LIN {X 0,Y 119.872,Z 1061.457,A -85,B 0,C 180,E1 -25663.563,E2 -25663.563} C_VEL
LIN {X 0,Y 121.874,Z 1058.966,A -85,B 0,C 180,E1 -25670.242,E2 -25670.242} C_VEL
LIN {X 0,Y 125.218,Z 1055.451,A -85,B 0,C 180,E1 -25676.679,E2 -25676.679} C_VEL
LIN {X 0,Y 129.866,Z 1050.86,A -85,B 0,C 180,E1 -25682.763,E2 -25682.763} C_VEL
LIN {X 0,Y 135.81,Z 1045.124,A -85,B 0,C 180,E1 -25688.387,E2 -25688.387} C_VEL
LIN {X 0,Y 141.031,Z 1040.06,A -85,B 0,C 180,E1 -25692.278,E2 -25692.278} C_VEL
LIN {X 0,Y 148.928,Z 1032.029,A -85,B 0,C 180,E1 -25697.007,E2 -25697.007} C_VEL
LIN {X 0,Y 151.068,Z 1029.838,A -85,B 0,C 180,E1 -25698.076,E2 -25698.076} C_VEL
LIN {X 0,Y 153.644,Z 1026.725,A -85,B 0,C 180,E1 -25699.683,E2 -25699.683} C_VEL
LIN {X 0,Y 156.483,Z 1021.432,A -85,B 0,C 180,E1 -25702.602,E2 -25702.602} C_VEL
LIN {X 0,Y 159.483,Z 1015.894,A -85,B 0,C 180,E1 -25705.377,E2 -25705.377} C_VEL
LIN {X 0,Y 162.214,Z 1012.21,A -85,B 0,C 180,E1 -25706.721,E2 -25706.721} C_VEL
LIN {X 0,Y 171.119,Z 1001.077,A -85,B 0,C 180,E1 -25709.594,E2 -25709.594} C_VEL
LIN {X 0,Y 180.348,Z 987.934,A -85,B 0,C 180,E1 -25712.119,E2 -25712.119} C_VEL
LIN {X 0,Y 187.112,Z 977.199,A -85,B 0,C 180,E1 -25713.732,E2 -25713.732} C_VEL
LIN {X 0,Y 193.609,Z 965.54,A -85,B 0,C 180,E1 -25715.158,E2 -25715.158} C_VEL
LIN {X 0,Y 199.505,Z 953.526,A -85,B 0,C 180,E1 -25716.331,E2 -25716.331} C_VEL
LIN {X 0,Y 204.688,Z 941.214,A -85,B 0,C 180,E1 -25717.329,E2 -25717.329} C_VEL
LIN {X 0,Y 209.238,Z 928.68,A -85,B 0,C 180,E1 -25718.103,E2 -25718.103} C_VEL
LIN {X 0,Y 213.187,Z 915.532,A -85,B 0,C 180,E1 -25718.738,E2 -25718.738} C_VEL
LIN {X 0,Y 216.353,Z 902.36,A -85,B 0,C 180,E1 -25719.211,E2 -25719.211} C_VEL
LIN {X 0,Y 218.607,Z 889.44,A -85,B 0,C 180,E1 -25719.615,E2 -25719.615} C_VEL
LIN {X 0,Y 221.458,Z 863.499,A -85,B 0,C 180,E1 -25720.238,E2 -25720.238} C_VEL
LIN {X 0,Y 225.126,Z 826.857,A -85,B 0,C 180,E1 -25721.038,E2 -25721.038} C_VEL
LIN {X 0,Y 223.867,Z 823.253,A -85,B 0,C 180,E1 -25722.353,E2 -25722.353} C_VEL
LIN {X 0,Y 221.348,Z 817.719,A -85,B 0,C 180,E1 -25725.167,E2 -25725.167} C_VEL
LIN {X 0,Y 219.032,Z 813.003,A -85,B 0,C 180,E1 -25728.334,E2 -25728.334} C_VEL
LIN {X 0,Y 217.674,Z 810.199,A -85,B 0,C 180,E1 -25730.709,E2 -25730.709} C_VEL
LIN {X 0,Y 216.21,Z 806.853,A -85,B 0,C 180,E1 -25734.403,E2 -25734.403} C_VEL
LIN {X 0,Y 215.341,Z 804.93,A -85,B 0,C 180,E1 -25739.999,E2 -25739.999} C_VEL
LIN {X 0,Y 216.416,Z 807.28,A -85,B 0,C 180,E1 -25746.643,E2 -25746.643} C_VEL
LIN {X 0,Y 218.274,Z 811.333,A -85,B 0,C 180,E1 -25750.797,E2 -25750.797} C_VEL
LIN {X 0,Y 220.254,Z 815.508,A -85,B 0,C 180,E1 -25753.845,E2 -25753.845} C_VEL
LIN {X 0,Y 222.437,Z 820.088,A -85,B 0,C 180,E1 -25756.52,E2 -25756.52} C_VEL
LIN {X 0,Y 226.001,Z 828.064,A -85,B 0,C 180,E1 -25760.109,E2 -25760.109} C_VEL
LIN {X 0,Y 234.508,Z 846.019,A -85,B 0,C 180,E1 -25766.47,E2 -25766.47} C_VEL
LIN {X 0,Y 241.894,Z 856.796,A -85,B 0,C 180,E1 -25770.446,E2 -25770.446} C_VEL
LIN {X 0,Y 249.216,Z 865.395,A -85,B 0,C 180,E1 -25773.663,E2 -25773.663} C_VEL
LIN {X 0,Y 263.908,Z 879.329,A -85,B 0,C 180,E1 -25778.879,E2 -25778.879} C_VEL
LIN {X 0,Y 280.399,Z 892.407,A -85,B 0,C 180,E1 -25783.707,E2 -25783.707} C_VEL
LIN {X 0,Y 288.067,Z 898.214,A -85,B 0,C 180,E1 -25786.03,E2 -25786.03} C_VEL
LIN {X 0,Y 295.771,Z 904.316,A -85,B 0,C 180,E1 -25788.563,E2 -25788.563} C_VEL
LIN {X 0,Y 302.153,Z 909.232,A -85,B 0,C 180,E1 -25790.793,E2 -25790.793} C_VEL
LIN {X 0,Y 308.739,Z 914.279,A -85,B 0,C 180,E1 -25793.23,E2 -25793.23} C_VEL
LIN {X 0,Y 315.739,Z 919.877,A -85,B 0,C 180,E1 -25796.013,E2 -25796.013} C_VEL
LIN {X 0,Y 322.198,Z 924.602,A -85,B 0,C 180,E1 -25798.709,E2 -25798.709} C_VEL
LIN {X 0,Y 327.662,Z 928.89,A -85,B 0,C 180,E1 -25801.207,E2 -25801.207} C_VEL
LIN {X 0,Y 332.858,Z 932.301,A -85,B 0,C 180,E1 -25803.68,E2 -25803.68} C_VEL
LIN {X 0,Y 337.92,Z 936.346,A -85,B 0,C 180,E1 -25806.391,E2 -25806.391} C_VEL
LIN {X 0,Y 341.187,Z 938.576,A -85,B 0,C 180,E1 -25808.237,E2 -25808.237} C_VEL
LIN {X 0,Y 345.175,Z 940.955,A -85,B 0,C 180,E1 -25810.656,E2 -25810.656} C_VEL
LIN {X 0,Y 348.889,Z 944.049,A -85,B 0,C 180,E1 -25813.398,E2 -25813.398} C_VEL
LIN {X 0,Y 352.119,Z 946.467,A -85,B 0,C 180,E1 -25816.143,E2 -25816.143} C_VEL
LIN {X 0,Y 354.613,Z 947.948,A -85,B 0,C 180,E1 -25818.569,E2 -25818.569} C_VEL
LIN {X 0,Y 356.684,Z 948.845,A -85,B 0,C 180,E1 -25820.931,E2 -25820.931} C_VEL
LIN {X 0,Y 358.262,Z 949.527,A -85,B 0,C 180,E1 -25823.241,E2 -25823.241} C_VEL
LIN {X 0,Y 359.416,Z 950.168,A -85,B 0,C 180,E1 -25825.741,E2 -25825.741} C_VEL
LIN {X 0,Y 360.008,Z 950.332,A -85,B 0,C 180,E1 -25827.762,E2 -25827.762} C_VEL
LIN {X 0,Y 360.177,Z 950.528,A -85,B 0,C 180,E1 -25830,E2 -25830} C_VEL
LIN {X 0,Y 359.997,Z 950.345,A -85,B 0,C 180,E1 -25832.238,E2 -25832.238} C_VEL
LIN {X 0,Y 359.347,Z 950.13,A -85,B 0,C 180,E1 -25834.487,E2 -25834.487} C_VEL
LIN {X 0,Y 358.254,Z 949.537,A -85,B 0,C 180,E1 -25836.759,E2 -25836.759} C_VEL
LIN {X 0,Y 356.317,Z 948.732,A -85,B 0,C 180,E1 -25839.534,E2 -25839.534} C_VEL
LIN {X 0,Y 353.687,Z 947.457,A -85,B 0,C 180,E1 -25842.357,E2 -25842.357} C_VEL
LIN {X 0,Y 350.683,Z 945.481,A -85,B 0,C 180,E1 -25845.101,E2 -25845.101} C_VEL
LIN {X 0,Y 347.397,Z 942.776,A -85,B 0,C 180,E1 -25847.758,E2 -25847.758} C_VEL
LIN {X 0,Y 345.062,Z 940.837,A -85,B 0,C 180,E1 -25849.424,E2 -25849.424} C_VEL
LIN {X 0,Y 340.899,Z 938.445,A -85,B 0,C 180,E1 -25851.919,E2 -25851.919} C_VEL
LIN {X 0,Y 335.973,Z 934.874,A -85,B 0,C 180,E1 -25854.67,E2 -25854.67} C_VEL
LIN {X 0,Y 331.95,Z 931.717,A -85,B 0,C 180,E1 -25856.77,E2 -25856.77} C_VEL
LIN {X 0,Y 326.642,Z 928.193,A -85,B 0,C 180,E1 -25859.257,E2 -25859.257} C_VEL
LIN {X 0,Y 321.431,Z 923.928,A -85,B 0,C 180,E1 -25861.612,E2 -25861.612} C_VEL
LIN {X 0,Y 315.122,Z 919.405,A -85,B 0,C 180,E1 -25864.246,E2 -25864.246} C_VEL
LIN {X 0,Y 308.228,Z 913.886,A -85,B 0,C 180,E1 -25866.956,E2 -25866.956} C_VEL
LIN {X 0,Y 301.28,Z 908.527,A -85,B 0,C 180,E1 -25869.526,E2 -25869.526} C_VEL
LIN {X 0,Y 293.033,Z 902.244,A -85,B 0,C 180,E1 -25872.355,E2 -25872.355} C_VEL
LIN {X 0,Y 285.39,Z 896.212,A -85,B 0,C 180,E1 -25874.804,E2 -25874.804} C_VEL
LIN {X 0,Y 277.485,Z 890.054,A -85,B 0,C 180,E1 -25877.129,E2 -25877.129} C_VEL
LIN {X 0,Y 260.289,Z 876.113,A -85,B 0,C 180,E1 -25882.304,E2 -25882.304} C_VEL
LIN {X 0,Y 245.574,Z 861.451,A -85,B 0,C 180,E1 -25887.859,E2 -25887.859} C_VEL
LIN {X 0,Y 236.109,Z 848.6,A -85,B 0,C 180,E1 -25892.585,E2 -25892.585} C_VEL
LIN {X 0,Y 229.351,Z 836.123,A -85,B 0,C 180,E1 -25897.047,E2 -25897.047} C_VEL
LIN {X 0,Y 225.272,Z 826.453,A -85,B 0,C 180,E1 -25900.562,E2 -25900.562} C_VEL
LIN {X 0,Y 222.055,Z 819.193,A -85,B 0,C 180,E1 -25903.923,E2 -25903.923} C_VEL
LIN {X 0,Y 219.545,Z 813.93,A -85,B 0,C 180,E1 -25907.169,E2 -25907.169} C_VEL
LIN {X 0,Y 217.7,Z 810.223,A -85,B 0,C 180,E1 -25910.258,E2 -25910.258} C_VEL
LIN {X 0,Y 216.231,Z 806.874,A -85,B 0,C 180,E1 -25913.937,E2 -25913.937} C_VEL
LIN {X 0,Y 215.343,Z 804.916,A -85,B 0,C 180,E1 -25920.001,E2 -25920.001} C_VEL
LIN {X 0,Y 216.419,Z 807.254,A -85,B 0,C 180,E1 -25926.234,E2 -25926.234} C_VEL
LIN {X 0,Y 218.227,Z 811.308,A -85,B 0,C 180,E1 -25930.32,E2 -25930.32} C_VEL
LIN {X 0,Y 220.263,Z 815.5,A -85,B 0,C 180,E1 -25933.446,E2 -25933.446} C_VEL
LIN {X 0,Y 222.63,Z 820.514,A -85,B 0,C 180,E1 -25936.329,E2 -25936.329} C_VEL
LIN {X 0,Y 224.668,Z 825.364,A -85,B 0,C 180,E1 -25938.478,E2 -25938.478} C_VEL
LIN {X 0,Y 225.131,Z 826.859,A -85,B 0,C 180,E1 -25938.966,E2 -25938.966} C_VEL
LIN {X 0,Y 218.965,Z 886.847,A -85,B 0,C 180,E1 -25940.304,E2 -25940.304} C_VEL
LIN {X 0,Y 216.625,Z 900.823,A -85,B 0,C 180,E1 -25940.721,E2 -25940.721} C_VEL
LIN {X 0,Y 213.711,Z 913.481,A -85,B 0,C 180,E1 -25941.177,E2 -25941.177} C_VEL
LIN {X 0,Y 210.403,Z 925.095,A -85,B 0,C 180,E1 -25941.723,E2 -25941.723} C_VEL
LIN {X 0,Y 206.205,Z 937.255,A -85,B 0,C 180,E1 -25942.412,E2 -25942.412} C_VEL
LIN {X 0,Y 201.74,Z 948.504,A -85,B 0,C 180,E1 -25943.249,E2 -25943.249} C_VEL
LIN {X 0,Y 196.547,Z 959.793,A -85,B 0,C 180,E1 -25944.247,E2 -25944.247} C_VEL
LIN {X 0,Y 189.982,Z 972.216,A -85,B 0,C 180,E1 -25945.62,E2 -25945.62} C_VEL
LIN {X 0,Y 183.571,Z 983.007,A -85,B 0,C 180,E1 -25947.114,E2 -25947.114} C_VEL
LIN {X 0,Y 176.625,Z 993.498,A -85,B 0,C 180,E1 -25948.912,E2 -25948.912} C_VEL
LIN {X 0,Y 169.789,Z 1002.756,A -85,B 0,C 180,E1 -25950.81,E2 -25950.81} C_VEL
LIN {X 0,Y 161.973,Z 1012.482,A -85,B 0,C 180,E1 -25953.36,E2 -25953.36} C_VEL
LIN {X 0,Y 153.784,Z 1021.759,A -85,B 0,C 180,E1 -25956.449,E2 -25956.449} C_VEL
LIN {X 0,Y 146.382,Z 1029.6,A -85,B 0,C 180,E1 -25959.811,E2 -25959.811} C_VEL
LIN {X 0,Y 139.819,Z 1036.028,A -85,B 0,C 180,E1 -25963.212,E2 -25963.212} C_VEL
LIN {X 0,Y 132.338,Z 1042.991,A -85,B 0,C 180,E1 -25968.031,E2 -25968.031} C_VEL
LIN {X 0,Y 126.903,Z 1047.949,A -85,B 0,C 180,E1 -25972.47,E2 -25972.47} C_VEL
LIN {X 0,Y 121.171,Z 1053.059,A -85,B 0,C 180,E1 -25978.534,E2 -25978.534} C_VEL
LIN {X 0,Y 116.802,Z 1057.074,A -85,B 0,C 180,E1 -25985.091,E2 -25985.091} C_VEL
LIN {X 0,Y 113.843,Z 1060.051,A -85,B 0,C 180,E1 -25992.021,E2 -25992.021} C_VEL
LIN {X 0,Y 112.903,Z 1061.249,A -85,B 0,C 180,E1 -25995.582,E2 -25995.582} C_VEL
LIN {X 0,Y 112.065,Z 1062.744,A -85,B 0,C 180,E1 -26002.795,E2 -26002.795} C_VEL
LIN {X 0,Y 112.249,Z 1063.253,A -85,B 0,C 180,E1 -26010,E2 -26010} C_VEL
LIN {X 0,Y 112.065,Z 1062.744,A -85,B 0,C 180,E1 -26017.205,E2 -26017.205} C_VEL
LIN {X 0,Y 112.903,Z 1061.249,A -85,B 0,C 180,E1 -26024.418,E2 -26024.418} C_VEL
LIN {X 0,Y 115.144,Z 1058.758,A -85,B 0,C 180,E1 -26031.482,E2 -26031.482} C_VEL
LIN {X 0,Y 118.822,Z 1055.243,A -85,B 0,C 180,E1 -26038.24,E2 -26038.24} C_VEL
LIN {X 0,Y 123.86,Z 1050.651,A -85,B 0,C 180,E1 -26044.569,E2 -26044.569} C_VEL
LIN {X 0,Y 130.236,Z 1044.916,A -85,B 0,C 180,E1 -26050.357,E2 -26050.357} C_VEL
LIN {X 0,Y 135.788,Z 1039.852,A -85,B 0,C 180,E1 -26054.323,E2 -26054.323} C_VEL
LIN {X 0,Y 144.122,Z 1031.821,A -85,B 0,C 180,E1 -26059.097,E2 -26059.097} C_VEL
LIN {X 0,Y 150.93,Z 1024.839,A -85,B 0,C 180,E1 -26062.333,E2 -26062.333} C_VEL
LIN {X 0,Y 158.185,Z 1016.875,A -85,B 0,C 180,E1 -26065.277,E2 -26065.277} C_VEL
LIN {X 0,Y 162.214,Z 1012.21,A -85,B 0,C 180,E1 -26066.721,E2 -26066.721} C_VEL
LIN {X 0,Y 165.01,Z 1008.46,A -85,B 0,C 180,E1 -26067.984,E2 -26067.984} C_VEL
LIN {X 0,Y 171.161,Z 996.951,A -85,B 0,C 180,E1 -26072.133,E2 -26072.133} C_VEL
LIN {X 0,Y 173.688,Z 992.786,A -85,B 0,C 180,E1 -26073.247,E2 -26073.247} C_VEL
LIN {X 0,Y 174.683,Z 991.347,A -85,B 0,C 180,E1 -26073.546,E2 -26073.546} C_VEL
LIN {X 0,Y 184.053,Z 976.992,A -85,B 0,C 180,E1 -26075.732,E2 -26075.732} C_VEL
LIN {X 0,Y 190.722,Z 965.334,A -85,B 0,C 180,E1 -26077.104,E2 -26077.104} C_VEL
LIN {X 0,Y 196.746,Z 953.319,A -85,B 0,C 180,E1 -26078.237,E2 -26078.237} C_VEL
LIN {X 0,Y 202.056,Z 941.008,A -85,B 0,C 180,E1 -26079.188,E2 -26079.188} C_VEL
LIN {X 0,Y 206.672,Z 928.546,A -85,B 0,C 180,E1 -26079.927,E2 -26079.927} C_VEL
LIN {X 0,Y 210.786,Z 915.068,A -85,B 0,C 180,E1 -26080.546,E2 -26080.546} C_VEL
LIN {X 0,Y 213.935,Z 902.154,A -85,B 0,C 180,E1 -26080.99,E2 -26080.99} C_VEL
LIN {X 0,Y 216.252,Z 889.095,A -85,B 0,C 180,E1 -26081.385,E2 -26081.385} C_VEL
LIN {X 0,Y 219.172,Z 863.149,A -85,B 0,C 180,E1 -26081.99,E2 -26081.99} C_VEL
LIN {X 0,Y 222.528,Z 830.426,A -85,B 0,C 180,E1 -26082.687,E2 -26082.687} C_VEL
LIN {X 0,Y 219.902,Z 824.244,A -85,B 0,C 180,E1 -26085.777,E2 -26085.777} C_VEL
LIN {X 0,Y 217.724,Z 819.607,A -85,B 0,C 180,E1 -26088.95,E2 -26088.95} C_VEL
LIN {X 0,Y 216.563,Z 817.029,A -85,B 0,C 180,E1 -26091.132,E2 -26091.132} C_VEL
LIN {X 0,Y 215.347,Z 813.917,A -85,B 0,C 180,E1 -26094.381,E2 -26094.381} C_VEL
LIN {X 0,Y 214.471,Z 812.018,A -85,B 0,C 180,E1 -26099.999,E2 -26099.999} C_VEL
LIN {X 0,Y 215.424,Z 814.232,A -85,B 0,C 180,E1 -26106.321,E2 -26106.321} C_VEL
LIN {X 0,Y 217.192,Z 818.331,A -85,B 0,C 180,E1 -26110.5,E2 -26110.5} C_VEL
LIN {X 0,Y 219.025,Z 822.389,A -85,B 0,C 180,E1 -26113.452,E2 -26113.452} C_VEL
LIN {X 0,Y 221.218,Z 827.323,A -85,B 0,C 180,E1 -26116.258,E2 -26116.258} C_VEL
LIN {X 0,Y 224.222,Z 834.474,A -85,B 0,C 180,E1 -26119.433,E2 -26119.433} C_VEL
LIN {X 0,Y 232.161,Z 851.924,A -85,B 0,C 180,E1 -26125.69,E2 -26125.69} C_VEL
LIN {X 0,Y 239.542,Z 862.987,A -85,B 0,C 180,E1 -26129.837,E2 -26129.837} C_VEL
LIN {X 0,Y 246.772,Z 871.64,A -85,B 0,C 180,E1 -26133.123,E2 -26133.123} C_VEL
LIN {X 0,Y 261.379,Z 885.809,A -85,B 0,C 180,E1 -26138.569,E2 -26138.569} C_VEL
LIN {X 0,Y 278.021,Z 899.242,A -85,B 0,C 180,E1 -26143.663,E2 -26143.663} C_VEL
LIN {X 0,Y 286.438,Z 905.644,A -85,B 0,C 180,E1 -26146.242,E2 -26146.242} C_VEL
LIN {X 0,Y 294.406,Z 911.893,A -85,B 0,C 180,E1 -26148.889,E2 -26148.889} C_VEL
LIN {X 0,Y 301.317,Z 917.251,A -85,B 0,C 180,E1 -26151.332,E2 -26151.332} C_VEL
LIN {X 0,Y 308.076,Z 922.37,A -85,B 0,C 180,E1 -26153.865,E2 -26153.865} C_VEL
LIN {X 0,Y 313.516,Z 926.694,A -85,B 0,C 180,E1 -26156.038,E2 -26156.038} C_VEL
LIN {X 0,Y 318.308,Z 930.045,A -85,B 0,C 180,E1 -26158.002,E2 -26158.002} C_VEL
LIN {X 0,Y 323.471,Z 934.316,A -85,B 0,C 180,E1 -26160.35,E2 -26160.35} C_VEL
LIN {X 0,Y 328.166,Z 937.554,A -85,B 0,C 180,E1 -26162.527,E2 -26162.527} C_VEL
LIN {X 0,Y 331.846,Z 940.152,A -85,B 0,C 180,E1 -26164.352,E2 -26164.352} C_VEL
LIN {X 0,Y 336.401,Z 943.645,A -85,B 0,C 180,E1 -26166.813,E2 -26166.813} C_VEL
LIN {X 0,Y 340.978,Z 946.623,A -85,B 0,C 180,E1 -26169.489,E2 -26169.489} C_VEL
LIN {X 0,Y 343.183,Z 947.844,A -85,B 0,C 180,E1 -26170.874,E2 -26170.874} C_VEL
LIN {X 0,Y 346.673,Z 950.908,A -85,B 0,C 180,E1 -26173.512,E2 -26173.512} C_VEL
LIN {X 0,Y 349.681,Z 953.11,A -85,B 0,C 180,E1 -26176.044,E2 -26176.044} C_VEL
LIN {X 0,Y 352.248,Z 954.621,A -85,B 0,C 180,E1 -26178.492,E2 -26178.492} C_VEL
LIN {X 0,Y 354.404,Z 955.544,A -85,B 0,C 180,E1 -26180.872,E2 -26180.872} C_VEL
LIN {X 0,Y 356.021,Z 956.264,A -85,B 0,C 180,E1 -26183.198,E2 -26183.198} C_VEL
LIN {X 0,Y 357.124,Z 956.847,A -85,B 0,C 180,E1 -26185.485,E2 -26185.485} C_VEL
LIN {X 0,Y 357.782,Z 957.076,A -85,B 0,C 180,E1 -26187.749,E2 -26187.749} C_VEL
LIN {X 0,Y 357.955,Z 957.242,A -85,B 0,C 180,E1 -26190,E2 -26190} C_VEL
LIN {X 0,Y 357.78,Z 957.072,A -85,B 0,C 180,E1 -26192.251,E2 -26192.251} C_VEL
LIN {X 0,Y 357.124,Z 956.859,A -85,B 0,C 180,E1 -26194.515,E2 -26194.515} C_VEL
LIN {X 0,Y 356.018,Z 956.276,A -85,B 0,C 180,E1 -26196.802,E2 -26196.802} C_VEL
LIN {X 0,Y 354.412,Z 955.526,A -85,B 0,C 180,E1 -26199.128,E2 -26199.128} C_VEL
LIN {X 0,Y 351.878,Z 954.486,A -85,B 0,C 180,E1 -26201.859,E2 -26201.859} C_VEL
LIN {X 0,Y 348.814,Z 952.491,A -85,B 0,C 180,E1 -26204.737,E2 -26204.737} C_VEL
LIN {X 0,Y 345.773,Z 950.173,A -85,B 0,C 180,E1 -26207.199,E2 -26207.199} C_VEL
LIN {X 0,Y 342.768,Z 947.557,A -85,B 0,C 180,E1 -26209.411,E2 -26209.411} C_VEL
LIN {X 0,Y 338.59,Z 945.171,A -85,B 0,C 180,E1 -26211.938,E2 -26211.938} C_VEL
LIN {X 0,Y 334.748,Z 942.407,A -85,B 0,C 180,E1 -26214.105,E2 -26214.105} C_VEL
LIN {X 0,Y 330.048,Z 938.65,A -85,B 0,C 180,E1 -26216.578,E2 -26216.578} C_VEL
LIN {X 0,Y 324.807,Z 935.24,A -85,B 0,C 180,E1 -26219.062,E2 -26219.062} C_VEL
LIN {X 0,Y 320.233,Z 931.721,A -85,B 0,C 180,E1 -26221.14,E2 -26221.14} C_VEL
LIN {X 0,Y 315.14,Z 927.885,A -85,B 0,C 180,E1 -26223.297,E2 -26223.297} C_VEL
LIN {X 0,Y 308.039,Z 922.396,A -85,B 0,C 180,E1 -26226.135,E2 -26226.135} C_VEL
LIN {X 0,Y 301.04,Z 917.043,A -85,B 0,C 180,E1 -26228.767,E2 -26228.767} C_VEL
LIN {X 0,Y 294.407,Z 911.863,A -85,B 0,C 180,E1 -26231.111,E2 -26231.111} C_VEL
LIN {X 0,Y 287.048,Z 906.125,A -85,B 0,C 180,E1 -26233.568,E2 -26233.568} C_VEL
LIN {X 0,Y 278.774,Z 899.825,A -85,B 0,C 180,E1 -26236.11,E2 -26236.11} C_VEL
LIN {X 0,Y 264.554,Z 888.397,A -85,B 0,C 180,E1 -26240.39,E2 -26240.39} C_VEL
LIN {X 0,Y 251.369,Z 876.513,A -85,B 0,C 180,E1 -26245.022,E2 -26245.022} C_VEL
LIN {X 0,Y 240.24,Z 863.952,A -85,B 0,C 180,E1 -26249.815,E2 -26249.815} C_VEL
LIN {X 0,Y 231.838,Z 851.383,A -85,B 0,C 180,E1 -26254.517,E2 -26254.517} C_VEL
LIN {X 0,Y 223.285,Z 832.242,A -85,B 0,C 180,E1 -26261.491,E2 -26261.491} C_VEL
LIN {X 0,Y 220.446,Z 825.494,A -85,B 0,C 180,E1 -26264.676,E2 -26264.676} C_VEL
LIN {X 0,Y 218.195,Z 820.499,A -85,B 0,C 180,E1 -26267.798,E2 -26267.798} C_VEL
LIN {X 0,Y 216.597,Z 817.051,A -85,B 0,C 180,E1 -26270.664,E2 -26270.664} C_VEL
LIN {X 0,Y 215.365,Z 813.967,A -85,B 0,C 180,E1 -26273.912,E2 -26273.912} C_VEL
LIN {X 0,Y 214.472,Z 812.006,A -85,B 0,C 180,E1 -26280.001,E2 -26280.001} C_VEL
LIN {X 0,Y 215.442,Z 814.27,A -85,B 0,C 180,E1 -26285.969,E2 -26285.969} C_VEL
LIN {X 0,Y 217.069,Z 818.125,A -85,B 0,C 180,E1 -26289.875,E2 -26289.875} C_VEL
LIN {X 0,Y 218.9,Z 822.146,A -85,B 0,C 180,E1 -26292.87,E2 -26292.87} C_VEL
LIN {X 0,Y 220.979,Z 826.741,A -85,B 0,C 180,E1 -26295.566,E2 -26295.566} C_VEL
LIN {X 0,Y 222.53,Z 830.49,A -85,B 0,C 180,E1 -26297.322,E2 -26297.322} C_VEL
LIN {X 0,Y 216.563,Z 886.918,A -85,B 0,C 180,E1 -26298.548,E2 -26298.548} C_VEL
LIN {X 0,Y 214.101,Z 901.172,A -85,B 0,C 180,E1 -26298.958,E2 -26298.958} C_VEL
LIN {X 0,Y 211.004,Z 914.201,A -85,B 0,C 180,E1 -26299.414,E2 -26299.414} C_VEL
LIN {X 0,Y 207.105,Z 927.281,A -85,B 0,C 180,E1 -26300.026,E2 -26300.026} C_VEL
LIN {X 0,Y 202.819,Z 939.028,A -85,B 0,C 180,E1 -26300.68,E2 -26300.68} C_VEL
LIN {X 0,Y 198.281,Z 949.972,A -85,B 0,C 180,E1 -26301.503,E2 -26301.503} C_VEL
LIN {X 0,Y 192.98,Z 961.024,A -85,B 0,C 180,E1 -26302.469,E2 -26302.469} C_VEL
LIN {X 0,Y 186.996,Z 972.009,A -85,B 0,C 180,E1 -26303.641,E2 -26303.641} C_VEL
LIN {X 0,Y 180.413,Z 982.8,A -85,B 0,C 180,E1 -26305.085,E2 -26305.085} C_VEL
LIN {X 0,Y 173.279,Z 993.291,A -85,B 0,C 180,E1 -26306.84,E2 -26306.84} C_VEL
LIN {X 0,Y 166.23,Z 1002.549,A -85,B 0,C 180,E1 -26308.687,E2 -26308.687} C_VEL
LIN {X 0,Y 158.135,Z 1012.274,A -85,B 0,C 180,E1 -26311.185,E2 -26311.185} C_VEL
LIN {X 0,Y 150.343,Z 1020.824,A -85,B 0,C 180,E1 -26313.959,E2 -26313.959} C_VEL
LIN {X 0,Y 141.866,Z 1029.391,A -85,B 0,C 180,E1 -26317.569,E2 -26317.569} C_VEL
LIN {X 0,Y 134.982,Z 1035.819,A -85,B 0,C 180,E1 -26320.98,E2 -26320.98} C_VEL
LIN {X 0,Y 126.504,Z 1043.245,A -85,B 0,C 180,E1 -26326.239,E2 -26326.239} C_VEL
LIN {X 0,Y 121.27,Z 1047.741,A -85,B 0,C 180,E1 -26330.397,E2 -26330.397} C_VEL
LIN {X 0,Y 115.076,Z 1052.85,A -85,B 0,C 180,E1 -26336.658,E2 -26336.658} C_VEL
LIN {X 0,Y 110.309,Z 1056.866,A -85,B 0,C 180,E1 -26343.514,E2 -26343.514} C_VEL
LIN {X 0,Y 107.051,Z 1059.843,A -85,B 0,C 180,E1 -26350.838,E2 -26350.838} C_VEL
LIN {X 0,Y 105.964,Z 1061.041,A -85,B 0,C 180,E1 -26354.616,E2 -26354.616} C_VEL
LIN {X 0,Y 104.997,Z 1062.538,A -85,B 0,C 180,E1 -26362.307,E2 -26362.307} C_VEL
LIN {X 0,Y 105.167,Z 1063.048,A -85,B 0,C 180,E1 -26370,E2 -26370} C_VEL
LIN {X 0,Y 104.997,Z 1062.538,A -85,B 0,C 180,E1 -26377.693,E2 -26377.693} C_VEL
LIN {X 0,Y 105.964,Z 1061.041,A -85,B 0,C 180,E1 -26385.384,E2 -26385.384} C_VEL
LIN {X 0,Y 108.476,Z 1058.55,A -85,B 0,C 180,E1 -26392.875,E2 -26392.875} C_VEL
LIN {X 0,Y 113.767,Z 1053.943,A -85,B 0,C 180,E1 -26401.673,E2 -26401.673} C_VEL
LIN {X 0,Y 117.986,Z 1050.442,A -85,B 0,C 180,E1 -26406.559,E2 -26406.559} C_VEL
LIN {X 0,Y 124.829,Z 1044.707,A -85,B 0,C 180,E1 -26412.5,E2 -26412.5} C_VEL
LIN {X 0,Y 130.73,Z 1039.643,A -85,B 0,C 180,E1 -26416.53,E2 -26416.53} C_VEL
LIN {X 0,Y 139.533,Z 1031.613,A -85,B 0,C 180,E1 -26421.323,E2 -26421.323} C_VEL
LIN {X 0,Y 146.643,Z 1024.63,A -85,B 0,C 180,E1 -26424.559,E2 -26424.559} C_VEL
LIN {X 0,Y 154.201,Z 1016.666,A -85,B 0,C 180,E1 -26427.474,E2 -26427.474} C_VEL
LIN {X 0,Y 162.114,Z 1007.559,A -85,B 0,C 180,E1 -26430.114,E2 -26430.114} C_VEL
LIN {X 0,Y 169.025,Z 999.002,A -85,B 0,C 180,E1 -26432.073,E2 -26432.073} C_VEL
LIN {X 0,Y 174.683,Z 991.347,A -85,B 0,C 180,E1 -26433.546,E2 -26433.546} C_VEL
LIN {X 0,Y 177.43,Z 987.024,A -85,B 0,C 180,E1 -26434.518,E2 -26434.518} C_VEL
LIN {X 0,Y 180.934,Z 979.913,A -85,B 0,C 180,E1 -26436.439,E2 -26436.439} C_VEL
LIN {X 0,Y 184.308,Z 972.446,A -85,B 0,C 180,E1 -26438.178,E2 -26438.178} C_VEL
LIN {X 0,Y 186.757,Z 967.576,A -85,B 0,C 180,E1 -26438.867,E2 -26438.867} C_VEL
LIN {X 0,Y 194.216,Z 953.113,A -85,B 0,C 180,E1 -26440.19,E2 -26440.19} C_VEL
LIN {X 0,Y 199.64,Z 940.802,A -85,B 0,C 180,E1 -26441.096,E2 -26441.096} C_VEL
LIN {X 0,Y 204.456,Z 927.989,A -85,B 0,C 180,E1 -26441.816,E2 -26441.816} C_VEL
LIN {X 0,Y 208.601,Z 914.56,A -85,B 0,C 180,E1 -26442.404,E2 -26442.404} C_VEL
LIN {X 0,Y 211.727,Z 901.949,A -85,B 0,C 180,E1 -26442.809,E2 -26442.809} C_VEL
LIN {X 0,Y 214.178,Z 888.237,A -85,B 0,C 180,E1 -26443.204,E2 -26443.204} C_VEL
LIN {X 0,Y 217.291,Z 860.999,A -85,B 0,C 180,E1 -26443.808,E2 -26443.808} C_VEL
LIN {X 0,Y 220.024,Z 834.599,A -85,B 0,C 180,E1 -26444.39,E2 -26444.39} C_VEL
LIN {X 0,Y 217.998,Z 829.679,A -85,B 0,C 180,E1 -26447.076,E2 -26447.076} C_VEL
LIN {X 0,Y 216.124,Z 825.463,A -85,B 0,C 180,E1 -26450.17,E2 -26450.17} C_VEL
LIN {X 0,Y 215.463,Z 823.859,A -85,B 0,C 180,E1 -26451.559,E2 -26451.559} C_VEL
LIN {X 0,Y 214.33,Z 820.833,A -85,B 0,C 180,E1 -26454.826,E2 -26454.826} C_VEL
LIN {X 0,Y 213.601,Z 819.102,A -85,B 0,C 180,E1 -26459.999,E2 -26459.999} C_VEL
LIN {X 0,Y 214.443,Z 821.151,A -85,B 0,C 180,E1 -26465.996,E2 -26465.996} C_VEL
LIN {X 0,Y 215.971,Z 824.994,A -85,B 0,C 180,E1 -26469.914,E2 -26469.914} C_VEL
LIN {X 0,Y 217.728,Z 829.107,A -85,B 0,C 180,E1 -26472.94,E2 -26472.94} C_VEL
LIN {X 0,Y 219.911,Z 834.326,A -85,B 0,C 180,E1 -26475.881,E2 -26475.881} C_VEL
LIN {X 0,Y 222.513,Z 841.064,A -85,B 0,C 180,E1 -26478.794,E2 -26478.794} C_VEL
LIN {X 0,Y 229.913,Z 857.92,A -85,B 0,C 180,E1 -26484.93,E2 -26484.93} C_VEL
LIN {X 0,Y 237.2,Z 869.156,A -85,B 0,C 180,E1 -26489.207,E2 -26489.207} C_VEL
LIN {X 0,Y 244.089,Z 877.707,A -85,B 0,C 180,E1 -26492.521,E2 -26492.521} C_VEL
LIN {X 0,Y 253.01,Z 886.872,A -85,B 0,C 180,E1 -26496.176,E2 -26496.176} C_VEL
LIN {X 0,Y 267.005,Z 899.353,A -85,B 0,C 180,E1 -26501.087,E2 -26501.087} C_VEL
LIN {X 0,Y 279.242,Z 908.885,A -85,B 0,C 180,E1 -26504.805,E2 -26504.805} C_VEL
LIN {X 0,Y 287.006,Z 914.912,A -85,B 0,C 180,E1 -26507.274,E2 -26507.274} C_VEL
LIN {X 0,Y 294.801,Z 920.847,A -85,B 0,C 180,E1 -26509.935,E2 -26509.935} C_VEL
LIN {X 0,Y 301.581,Z 926.116,A -85,B 0,C 180,E1 -26512.403,E2 -26512.403} C_VEL
LIN {X 0,Y 306.464,Z 929.948,A -85,B 0,C 180,E1 -26514.28,E2 -26514.28} C_VEL
LIN {X 0,Y 311.921,Z 934.137,A -85,B 0,C 180,E1 -26516.475,E2 -26516.475} C_VEL
LIN {X 0,Y 317.061,Z 937.919,A -85,B 0,C 180,E1 -26518.637,E2 -26518.637} C_VEL
LIN {X 0,Y 323.208,Z 942.601,A -85,B 0,C 180,E1 -26521.421,E2 -26521.421} C_VEL
LIN {X 0,Y 326.949,Z 945.025,A -85,B 0,C 180,E1 -26523.167,E2 -26523.167} C_VEL
LIN {X 0,Y 332.929,Z 949.682,A -85,B 0,C 180,E1 -26526.355,E2 -26526.355} C_VEL
LIN {X 0,Y 335.634,Z 951.499,A -85,B 0,C 180,E1 -26527.858,E2 -26527.858} C_VEL
LIN {X 0,Y 340.34,Z 954.293,A -85,B 0,C 180,E1 -26530.708,E2 -26530.708} C_VEL
LIN {X 0,Y 344.248,Z 957.66,A -85,B 0,C 180,E1 -26533.641,E2 -26533.641} C_VEL
LIN {X 0,Y 347.325,Z 959.859,A -85,B 0,C 180,E1 -26536.228,E2 -26536.228} C_VEL
LIN {X 0,Y 349.561,Z 961.172,A -85,B 0,C 180,E1 -26538.402,E2 -26538.402} C_VEL
LIN {X 0,Y 351.697,Z 962.089,A -85,B 0,C 180,E1 -26540.801,E2 -26540.801} C_VEL
LIN {X 0,Y 353.587,Z 962.944,A -85,B 0,C 180,E1 -26543.617,E2 -26543.617} C_VEL
LIN {X 0,Y 354.44,Z 963.397,A -85,B 0,C 180,E1 -26545.451,E2 -26545.451} C_VEL
LIN {X 0,Y 355.128,Z 963.663,A -85,B 0,C 180,E1 -26547.732,E2 -26547.732} C_VEL
LIN {X 0,Y 355.301,Z 963.827,A -85,B 0,C 180,E1 -26550,E2 -26550} C_VEL
LIN {X 0,Y 355.124,Z 963.659,A -85,B 0,C 180,E1 -26552.268,E2 -26552.268} C_VEL
LIN {X 0,Y 354.438,Z 963.407,A -85,B 0,C 180,E1 -26554.549,E2 -26554.549} C_VEL
LIN {X 0,Y 353.291,Z 962.834,A -85,B 0,C 180,E1 -26556.855,E2 -26556.855} C_VEL
LIN {X 0,Y 351.692,Z 962.071,A -85,B 0,C 180,E1 -26559.199,E2 -26559.199} C_VEL
LIN {X 0,Y 349.539,Z 961.213,A -85,B 0,C 180,E1 -26561.599,E2 -26561.599} C_VEL
LIN {X 0,Y 346.986,Z 959.635,A -85,B 0,C 180,E1 -26564.066,E2 -26564.066} C_VEL
LIN {X 0,Y 343.909,Z 957.33,A -85,B 0,C 180,E1 -26566.624,E2 -26566.624} C_VEL
LIN {X 0,Y 340.329,Z 954.258,A -85,B 0,C 180,E1 -26569.293,E2 -26569.293} C_VEL
LIN {X 0,Y 335.619,Z 951.534,A -85,B 0,C 180,E1 -26572.143,E2 -26572.143} C_VEL
LIN {X 0,Y 331.686,Z 948.69,A -85,B 0,C 180,E1 -26574.342,E2 -26574.342} C_VEL
LIN {X 0,Y 326.904,Z 944.921,A -85,B 0,C 180,E1 -26576.837,E2 -26576.837} C_VEL
LIN {X 0,Y 321.905,Z 941.677,A -85,B 0,C 180,E1 -26579.157,E2 -26579.157} C_VEL
LIN {X 0,Y 317.017,Z 937.921,A -85,B 0,C 180,E1 -26581.377,E2 -26581.377} C_VEL
LIN {X 0,Y 314.625,Z 935.976,A -85,B 0,C 180,E1 -26582.418,E2 -26582.418} C_VEL
LIN {X 0,Y 308.492,Z 931.56,A -85,B 0,C 180,E1 -26584.902,E2 -26584.902} C_VEL
LIN {X 0,Y 301.599,Z 926.068,A -85,B 0,C 180,E1 -26587.602,E2 -26587.602} C_VEL
LIN {X 0,Y 294.435,Z 920.518,A -85,B 0,C 180,E1 -26590.199,E2 -26590.199} C_VEL
LIN {X 0,Y 286.965,Z 914.952,A -85,B 0,C 180,E1 -26592.717,E2 -26592.717} C_VEL
LIN {X 0,Y 279.265,Z 908.834,A -85,B 0,C 180,E1 -26595.2,E2 -26595.2} C_VEL
LIN {X 0,Y 266.015,Z 898.545,A -85,B 0,C 180,E1 -26599.228,E2 -26599.228} C_VEL
LIN {X 0,Y 253.459,Z 887.287,A -85,B 0,C 180,E1 -26603.652,E2 -26603.652} C_VEL
LIN {X 0,Y 245.843,Z 879.514,A -85,B 0,C 180,E1 -26606.735,E2 -26606.735} C_VEL
LIN {X 0,Y 238.031,Z 870.328,A -85,B 0,C 180,E1 -26610.364,E2 -26610.364} C_VEL
LIN {X 0,Y 229.808,Z 857.754,A -85,B 0,C 180,E1 -26615.139,E2 -26615.139} C_VEL
LIN {X 0,Y 222.52,Z 841.016,A -85,B 0,C 180,E1 -26621.206,E2 -26621.206} C_VEL
LIN {X 0,Y 219.626,Z 833.66,A -85,B 0,C 180,E1 -26624.467,E2 -26624.467} C_VEL
LIN {X 0,Y 217.652,Z 828.934,A -85,B 0,C 180,E1 -26627.174,E2 -26627.174} C_VEL
LIN {X 0,Y 215.719,Z 824.3,A -85,B 0,C 180,E1 -26630.625,E2 -26630.625} C_VEL
LIN {X 0,Y 214.351,Z 820.85,A -85,B 0,C 180,E1 -26634.356,E2 -26634.356} C_VEL
LIN {X 0,Y 213.601,Z 819.104,A -85,B 0,C 180,E1 -26640.001,E2 -26640.001} C_VEL
LIN {X 0,Y 214.422,Z 821.124,A -85,B 0,C 180,E1 -26645.526,E2 -26645.526} C_VEL
LIN {X 0,Y 215.953,Z 825.012,A -85,B 0,C 180,E1 -26649.483,E2 -26649.483} C_VEL
LIN {X 0,Y 217.706,Z 829.079,A -85,B 0,C 180,E1 -26652.502,E2 -26652.502} C_VEL
LIN {X 0,Y 219.72,Z 833.891,A -85,B 0,C 180,E1 -26655.243,E2 -26655.243} C_VEL
LIN {X 0,Y 220.049,Z 834.669,A -85,B 0,C 180,E1 -26655.642,E2 -26655.642} C_VEL
LIN {X 0,Y 214.339,Z 887.197,A -85,B 0,C 180,E1 -26656.758,E2 -26656.758} C_VEL
LIN {X 0,Y 211.674,Z 902.086,A -85,B 0,C 180,E1 -26657.174,E2 -26657.174} C_VEL
LIN {X 0,Y 207.454,Z 918.889,A -85,B 0,C 180,E1 -26657.765,E2 -26657.765} C_VEL
LIN {X 0,Y 201.909,Z 935.062,A -85,B 0,C 180,E1 -26658.55,E2 -26658.55} C_VEL
LIN {X 0,Y 196.546,Z 948.091,A -85,B 0,C 180,E1 -26659.425,E2 -26659.425} C_VEL
LIN {X 0,Y 191.135,Z 959.38,A -85,B 0,C 180,E1 -26660.347,E2 -26660.347} C_VEL
LIN {X 0,Y 184.254,Z 971.803,A -85,B 0,C 180,E1 -26661.61,E2 -26661.61} C_VEL
LIN {X 0,Y 177.489,Z 982.592,A -85,B 0,C 180,E1 -26662.986,E2 -26662.986} C_VEL
LIN {X 0,Y 170.161,Z 993.083,A -85,B 0,C 180,E1 -26664.685,E2 -26664.685} C_VEL
LIN {X 0,Y 162.924,Z 1002.342,A -85,B 0,C 180,E1 -26666.484,E2 -26666.484} C_VEL
LIN {X 0,Y 154.526,Z 1012.066,A -85,B 0,C 180,E1 -26668.897,E2 -26668.897} C_VEL
LIN {X 0,Y 145.41,Z 1021.621,A -85,B 0,C 180,E1 -26671.997,E2 -26671.997} C_VEL
LIN {X 0,Y 137.581,Z 1029.182,A -85,B 0,C 180,E1 -26675.185,E2 -26675.185} C_VEL
LIN {X 0,Y 130.361,Z 1035.61,A -85,B 0,C 180,E1 -26678.584,E2 -26678.584} C_VEL
LIN {X 0,Y 121.903,Z 1042.645,A -85,B 0,C 180,E1 -26683.556,E2 -26683.556} C_VEL
LIN {X 0,Y 115.796,Z 1047.532,A -85,B 0,C 180,E1 -26688.118,E2 -26688.118} C_VEL
LIN {X 0,Y 109.131,Z 1052.641,A -85,B 0,C 180,E1 -26694.579,E2 -26694.579} C_VEL
LIN {X 0,Y 103.924,Z 1056.658,A -85,B 0,C 180,E1 -26701.747,E2 -26701.747} C_VEL
LIN {X 0,Y 100.285,Z 1059.635,A -85,B 0,C 180,E1 -26709.489,E2 -26709.489} C_VEL
LIN {X 0,Y 99.062,Z 1060.833,A -85,B 0,C 180,E1 -26713.514,E2 -26713.514} C_VEL
LIN {X 0,Y 97.923,Z 1062.331,A -85,B 0,C 180,E1 -26721.747,E2 -26721.747} C_VEL
LIN {X 0,Y 98.073,Z 1062.843,A -85,B 0,C 180,E1 -26730,E2 -26730} C_VEL
LIN {X 0,Y 97.923,Z 1062.331,A -85,B 0,C 180,E1 -26738.253,E2 -26738.253} C_VEL
LIN {X 0,Y 99.062,Z 1060.833,A -85,B 0,C 180,E1 -26746.486,E2 -26746.486} C_VEL
LIN {X 0,Y 101.886,Z 1058.342,A -85,B 0,C 180,E1 -26754.448,E2 -26754.448} C_VEL
LIN {X 0,Y 107.697,Z 1053.734,A -85,B 0,C 180,E1 -26763.688,E2 -26763.688} C_VEL
LIN {X 0,Y 112.27,Z 1050.233,A -85,B 0,C 180,E1 -26768.754,E2 -26768.754} C_VEL
LIN {X 0,Y 119.593,Z 1044.498,A -85,B 0,C 180,E1 -26774.843,E2 -26774.843} C_VEL
LIN {X 0,Y 125.881,Z 1039.435,A -85,B 0,C 180,E1 -26778.911,E2 -26778.911} C_VEL
LIN {X 0,Y 135.152,Z 1031.405,A -85,B 0,C 180,E1 -26783.706,E2 -26783.706} C_VEL
LIN {X 0,Y 142.593,Z 1024.422,A -85,B 0,C 180,E1 -26786.915,E2 -26786.915} C_VEL
LIN {X 0,Y 150.465,Z 1016.459,A -85,B 0,C 180,E1 -26789.778,E2 -26789.778} C_VEL
LIN {X 0,Y 158.653,Z 1007.351,A -85,B 0,C 180,E1 -26792.367,E2 -26792.367} C_VEL
LIN {X 0,Y 165.795,Z 998.795,A -85,B 0,C 180,E1 -26794.258,E2 -26794.258} C_VEL
LIN {X 0,Y 173.64,Z 988.236,A -85,B 0,C 180,E1 -26796.169,E2 -26796.169} C_VEL
LIN {X 0,Y 181.235,Z 976.785,A -85,B 0,C 180,E1 -26797.791,E2 -26797.791} C_VEL
LIN {X 0,Y 186.757,Z 967.576,A -85,B 0,C 180,E1 -26798.867,E2 -26798.867} C_VEL
LIN {X 0,Y 189.16,Z 962.64,A -85,B 0,C 180,E1 -26799.528,E2 -26799.528} C_VEL
LIN {X 0,Y 195.169,Z 946.544,A -85,B 0,C 180,E1 -26802.488,E2 -26802.488} C_VEL
LIN {X 0,Y 197.179,Z 941.269,A -85,B 0,C 180,E1 -26803.011,E2 -26803.011} C_VEL
LIN {X 0,Y 202.263,Z 928.049,A -85,B 0,C 180,E1 -26803.715,E2 -26803.715} C_VEL
LIN {X 0,Y 206.485,Z 914.65,A -85,B 0,C 180,E1 -26804.272,E2 -26804.272} C_VEL
LIN {X 0,Y 209.822,Z 901.345,A -85,B 0,C 180,E1 -26804.671,E2 -26804.671} C_VEL
LIN {X 0,Y 212.106,Z 888.938,A -85,B 0,C 180,E1 -26805.021,E2 -26805.021} C_VEL
LIN {X 0,Y 215.082,Z 863.886,A -85,B 0,C 180,E1 -26805.565,E2 -26805.565} C_VEL
LIN {X 0,Y 217.729,Z 839.039,A -85,B 0,C 180,E1 -26806.085,E2 -26806.085} C_VEL
LIN {X 0,Y 215.989,Z 834.722,A -85,B 0,C 180,E1 -26808.741,E2 -26808.741} C_VEL
LIN {X 0,Y 214.378,Z 830.67,A -85,B 0,C 180,E1 -26811.991,E2 -26811.991} C_VEL
LIN {X 0,Y 213.324,Z 827.767,A -85,B 0,C 180,E1 -26815.275,E2 -26815.275} C_VEL
LIN {X 0,Y 212.733,Z 826.172,A -85,B 0,C 180,E1 -26819.999,E2 -26819.999} C_VEL
LIN {X 0,Y 213.461,Z 828.133,A -85,B 0,C 180,E1 -26825.668,E2 -26825.668} C_VEL
LIN {X 0,Y 214.817,Z 831.746,A -85,B 0,C 180,E1 -26829.414,E2 -26829.414} C_VEL
LIN {X 0,Y 216.163,Z 835.121,A -85,B 0,C 180,E1 -26831.955,E2 -26831.955} C_VEL
LIN {X 0,Y 217.688,Z 838.959,A -85,B 0,C 180,E1 -26834.269,E2 -26834.269} C_VEL
LIN {X 0,Y 220.468,Z 846.461,A -85,B 0,C 180,E1 -26837.724,E2 -26837.724} C_VEL
LIN {X 0,Y 227.576,Z 863.681,A -85,B 0,C 180,E1 -26844.064,E2 -26844.064} C_VEL
LIN {X 0,Y 234.798,Z 875.231,A -85,B 0,C 180,E1 -26848.53,E2 -26848.53} C_VEL
LIN {X 0,Y 241.82,Z 884.198,A -85,B 0,C 180,E1 -26852.094,E2 -26852.094} C_VEL
LIN {X 0,Y 254.007,Z 896.975,A -85,B 0,C 180,E1 -26857.323,E2 -26857.323} C_VEL
LIN {X 0,Y 271.493,Z 911.694,A -85,B 0,C 180,E1 -26863.313,E2 -26863.313} C_VEL
LIN {X 0,Y 279.915,Z 918.129,A -85,B 0,C 180,E1 -26865.912,E2 -26865.912} C_VEL
LIN {X 0,Y 287.101,Z 923.78,A -85,B 0,C 180,E1 -26868.297,E2 -26868.297} C_VEL
LIN {X 0,Y 292.641,Z 928.016,A -85,B 0,C 180,E1 -26870.219,E2 -26870.219} C_VEL
LIN {X 0,Y 299.848,Z 933.462,A -85,B 0,C 180,E1 -26872.835,E2 -26872.835} C_VEL
LIN {X 0,Y 306.733,Z 938.969,A -85,B 0,C 180,E1 -26875.572,E2 -26875.572} C_VEL
LIN {X 0,Y 313.585,Z 943.984,A -85,B 0,C 180,E1 -26878.39,E2 -26878.39} C_VEL
LIN {X 0,Y 319.445,Z 948.489,A -85,B 0,C 180,E1 -26881.053,E2 -26881.053} C_VEL
LIN {X 0,Y 323.553,Z 951.205,A -85,B 0,C 180,E1 -26882.944,E2 -26882.944} C_VEL
LIN {X 0,Y 329.516,Z 955.81,A -85,B 0,C 180,E1 -26886.095,E2 -26886.095} C_VEL
LIN {X 0,Y 333.175,Z 958.268,A -85,B 0,C 180,E1 -26888.144,E2 -26888.144} C_VEL
LIN {X 0,Y 337.104,Z 960.59,A -85,B 0,C 180,E1 -26890.515,E2 -26890.515} C_VEL
LIN {X 0,Y 340.766,Z 963.685,A -85,B 0,C 180,E1 -26893.218,E2 -26893.218} C_VEL
LIN {X 0,Y 343.898,Z 965.996,A -85,B 0,C 180,E1 -26895.805,E2 -26895.805} C_VEL
LIN {X 0,Y 346.507,Z 967.575,A -85,B 0,C 180,E1 -26898.298,E2 -26898.298} C_VEL
LIN {X 0,Y 348.821,Z 968.56,A -85,B 0,C 180,E1 -26900.835,E2 -26900.835} C_VEL
LIN {X 0,Y 350.384,Z 969.296,A -85,B 0,C 180,E1 -26903.088,E2 -26903.088} C_VEL
LIN {X 0,Y 351.566,Z 969.87,A -85,B 0,C 180,E1 -26905.414,E2 -26905.414} C_VEL
LIN {X 0,Y 352.282,Z 970.169,A -85,B 0,C 180,E1 -26907.713,E2 -26907.713} C_VEL
LIN {X 0,Y 352.467,Z 970.314,A -85,B 0,C 180,E1 -26910,E2 -26910} C_VEL
LIN {X 0,Y 352.279,Z 970.166,A -85,B 0,C 180,E1 -26912.287,E2 -26912.287} C_VEL
LIN {X 0,Y 351.555,Z 969.895,A -85,B 0,C 180,E1 -26914.586,E2 -26914.586} C_VEL
LIN {X 0,Y 350.374,Z 969.305,A -85,B 0,C 180,E1 -26916.912,E2 -26916.912} C_VEL
LIN {X 0,Y 348.714,Z 968.517,A -85,B 0,C 180,E1 -26919.278,E2 -26919.278} C_VEL
LIN {X 0,Y 346.492,Z 967.595,A -85,B 0,C 180,E1 -26921.702,E2 -26921.702} C_VEL
LIN {X 0,Y 343.901,Z 965.989,A -85,B 0,C 180,E1 -26924.195,E2 -26924.195} C_VEL
LIN {X 0,Y 340.787,Z 963.639,A -85,B 0,C 180,E1 -26926.781,E2 -26926.781} C_VEL
LIN {X 0,Y 337.101,Z 960.567,A -85,B 0,C 180,E1 -26929.485,E2 -26929.485} C_VEL
LIN {X 0,Y 332.252,Z 957.698,A -85,B 0,C 180,E1 -26932.379,E2 -26932.379} C_VEL
LIN {X 0,Y 328.213,Z 954.776,A -85,B 0,C 180,E1 -26934.616,E2 -26934.616} C_VEL
LIN {X 0,Y 323.539,Z 951.101,A -85,B 0,C 180,E1 -26937.051,E2 -26937.051} C_VEL
LIN {X 0,Y 319.419,Z 948.474,A -85,B 0,C 180,E1 -26938.95,E2 -26938.95} C_VEL
LIN {X 0,Y 315.263,Z 945.371,A -85,B 0,C 180,E1 -26940.845,E2 -26940.845} C_VEL
LIN {X 0,Y 310.188,Z 941.451,A -85,B 0,C 180,E1 -26943.039,E2 -26943.039} C_VEL
LIN {X 0,Y 304.82,Z 937.492,A -85,B 0,C 180,E1 -26945.197,E2 -26945.197} C_VEL
LIN {X 0,Y 299.824,Z 933.441,A -85,B 0,C 180,E1 -26947.159,E2 -26947.159} C_VEL
LIN {X 0,Y 294.454,Z 929.432,A -85,B 0,C 180,E1 -26949.132,E2 -26949.132} C_VEL
LIN {X 0,Y 288.992,Z 925.145,A -85,B 0,C 180,E1 -26951.073,E2 -26951.073} C_VEL
LIN {X 0,Y 281.393,Z 919.379,A -85,B 0,C 180,E1 -26953.591,E2 -26953.591} C_VEL
LIN {X 0,Y 274.093,Z 913.737,A -85,B 0,C 180,E1 -26955.884,E2 -26955.884} C_VEL
LIN {X 0,Y 255.325,Z 898.205,A -85,B 0,C 180,E1 -26962.172,E2 -26962.172} C_VEL
LIN {X 0,Y 243.419,Z 885.997,A -85,B 0,C 180,E1 -26967.156,E2 -26967.156} C_VEL
LIN {X 0,Y 235.616,Z 876.432,A -85,B 0,C 180,E1 -26971.015,E2 -26971.015} C_VEL
LIN {X 0,Y 227.769,Z 864.05,A -85,B 0,C 180,E1 -26975.799,E2 -26975.799} C_VEL
LIN {X 0,Y 220.977,Z 848.047,A -85,B 0,C 180,E1 -26981.699,E2 -26981.699} C_VEL
LIN {X 0,Y 219.093,Z 842.774,A -85,B 0,C 180,E1 -26983.879,E2 -26983.879} C_VEL
LIN {X 0,Y 216.969,Z 837.088,A -85,B 0,C 180,E1 -26986.776,E2 -26986.776} C_VEL
LIN {X 0,Y 215.136,Z 832.607,A -85,B 0,C 180,E1 -26989.911,E2 -26989.911} C_VEL
LIN {X 0,Y 214.209,Z 830.329,A -85,B 0,C 180,E1 -26991.985,E2 -26991.985} C_VEL
LIN {X 0,Y 213.348,Z 827.745,A -85,B 0,C 180,E1 -26994.803,E2 -26994.803} C_VEL
LIN {X 0,Y 212.73,Z 826.199,A -85,B 0,C 180,E1 -27000.001,E2 -27000.001} C_VEL
LIN {X 0,Y 213.444,Z 828.08,A -85,B 0,C 180,E1 -27005.196,E2 -27005.196} C_VEL
LIN {X 0,Y 214.781,Z 831.715,A -85,B 0,C 180,E1 -27008.942,E2 -27008.942} C_VEL
LIN {X 0,Y 216.324,Z 835.548,A -85,B 0,C 180,E1 -27011.817,E2 -27011.817} C_VEL
LIN {X 0,Y 217.728,Z 839.029,A -85,B 0,C 180,E1 -27013.913,E2 -27013.913} C_VEL
LIN {X 0,Y 212.514,Z 886.282,A -85,B 0,C 180,E1 -27014.914,E2 -27014.914} C_VEL
LIN {X 0,Y 210.117,Z 899.781,A -85,B 0,C 180,E1 -27015.262,E2 -27015.262} C_VEL
LIN {X 0,Y 207.292,Z 911.675,A -85,B 0,C 180,E1 -27015.627,E2 -27015.627} C_VEL
LIN {X 0,Y 203.974,Z 922.985,A -85,B 0,C 180,E1 -27016.064,E2 -27016.064} C_VEL
LIN {X 0,Y 199.663,Z 935.091,A -85,B 0,C 180,E1 -27016.627,E2 -27016.627} C_VEL
LIN {X 0,Y 194.291,Z 947.884,A -85,B 0,C 180,E1 -27017.441,E2 -27017.441} C_VEL
LIN {X 0,Y 187.991,Z 960.611,A -85,B 0,C 180,E1 -27018.448,E2 -27018.448} C_VEL
LIN {X 0,Y 181.752,Z 971.597,A -85,B 0,C 180,E1 -27019.523,E2 -27019.523} C_VEL
LIN {X 0,Y 174.825,Z 982.386,A -85,B 0,C 180,E1 -27020.832,E2 -27020.832} C_VEL
LIN {X 0,Y 167.292,Z 992.876,A -85,B 0,C 180,E1 -27022.451,E2 -27022.451} C_VEL
LIN {X 0,Y 159.872,Z 1002.136,A -85,B 0,C 180,E1 -27024.196,E2 -27024.196} C_VEL
LIN {X 0,Y 151.192,Z 1011.858,A -85,B 0,C 180,E1 -27026.519,E2 -27026.519} C_VEL
LIN {X 0,Y 142.909,Z 1020.312,A -85,B 0,C 180,E1 -27029.132,E2 -27029.132} C_VEL
LIN {X 0,Y 133.565,Z 1028.974,A -85,B 0,C 180,E1 -27032.661,E2 -27032.661} C_VEL
LIN {X 0,Y 125.996,Z 1035.402,A -85,B 0,C 180,E1 -27036.023,E2 -27036.023} C_VEL
LIN {X 0,Y 116.75,Z 1042.66,A -85,B 0,C 180,E1 -27041.188,E2 -27041.188} C_VEL
LIN {X 0,Y 110.518,Z 1047.323,A -85,B 0,C 180,E1 -27045.614,E2 -27045.614} C_VEL
LIN {X 0,Y 103.323,Z 1052.432,A -85,B 0,C 180,E1 -27052.254,E2 -27052.254} C_VEL
LIN {X 0,Y 97.553,Z 1056.488,A -85,B 0,C 180,E1 -27059.828,E2 -27059.828} C_VEL
LIN {X 0,Y 93.589,Z 1059.427,A -85,B 0,C 180,E1 -27067.947,E2 -27067.947} C_VEL
LIN {X 0,Y 92.2,Z 1060.626,A -85,B 0,C 180,E1 -27072.248,E2 -27072.248} C_VEL
LIN {X 0,Y 90.852,Z 1062.124,A -85,B 0,C 180,E1 -27081.1,E2 -27081.1} C_VEL
LIN {X 0,Y 90.971,Z 1062.637,A -85,B 0,C 180,E1 -27090,E2 -27090} C_VEL
LIN {X 0,Y 90.852,Z 1062.124,A -85,B 0,C 180,E1 -27098.9,E2 -27098.9} C_VEL
LIN {X 0,Y 92.2,Z 1060.626,A -85,B 0,C 180,E1 -27107.752,E2 -27107.752} C_VEL
LIN {X 0,Y 95.39,Z 1058.134,A -85,B 0,C 180,E1 -27116.234,E2 -27116.234} C_VEL
LIN {X 0,Y 101.771,Z 1053.525,A -85,B 0,C 180,E1 -27125.942,E2 -27125.942} C_VEL
LIN {X 0,Y 106.743,Z 1050.025,A -85,B 0,C 180,E1 -27131.177,E2 -27131.177} C_VEL
LIN {X 0,Y 114.58,Z 1044.288,A -85,B 0,C 180,E1 -27137.394,E2 -27137.394} C_VEL
LIN {X 0,Y 121.259,Z 1039.226,A -85,B 0,C 180,E1 -27141.482,E2 -27141.482} C_VEL
LIN {X 0,Y 131.031,Z 1031.197,A -85,B 0,C 180,E1 -27146.237,E2 -27146.237} C_VEL
LIN {X 0,Y 138.792,Z 1024.214,A -85,B 0,C 180,E1 -27149.407,E2 -27149.407} C_VEL
LIN {X 0,Y 146.974,Z 1016.251,A -85,B 0,C 180,E1 -27152.204,E2 -27152.204} C_VEL
LIN {X 0,Y 155.444,Z 1007.143,A -85,B 0,C 180,E1 -27154.719,E2 -27154.719} C_VEL
LIN {X 0,Y 162.812,Z 998.587,A -85,B 0,C 180,E1 -27156.528,E2 -27156.528} C_VEL
LIN {X 0,Y 171.504,Z 987.14,A -85,B 0,C 180,E1 -27158.486,E2 -27158.486} C_VEL
LIN {X 0,Y 178.652,Z 976.578,A -85,B 0,C 180,E1 -27159.916,E2 -27159.916} C_VEL
LIN {X 0,Y 185.638,Z 964.921,A -85,B 0,C 180,E1 -27161.163,E2 -27161.163} C_VEL
LIN {X 0,Y 191.918,Z 952.907,A -85,B 0,C 180,E1 -27162.192,E2 -27162.192} C_VEL
LIN {X 0,Y 197.179,Z 941.269,A -85,B 0,C 180,E1 -27163.011,E2 -27163.011} C_VEL
LIN {X 0,Y 199.176,Z 935.93,A -85,B 0,C 180,E1 -27163.483,E2 -27163.483} C_VEL
LIN {X 0,Y 201.496,Z 927.302,A -85,B 0,C 180,E1 -27164.732,E2 -27164.732} C_VEL
LIN {X 0,Y 203.717,Z 918.527,A -85,B 0,C 180,E1 -27165.868,E2 -27165.868} C_VEL
LIN {X 0,Y 205.083,Z 912.964,A -85,B 0,C 180,E1 -27166.231,E2 -27166.231} C_VEL
LIN {X 0,Y 208.174,Z 900.552,A -85,B 0,C 180,E1 -27166.578,E2 -27166.578} C_VEL
LIN {X 0,Y 210.583,Z 887.271,A -85,B 0,C 180,E1 -27166.929,E2 -27166.929} C_VEL
LIN {X 0,Y 214.414,Z 854.682,A -85,B 0,C 180,E1 -27167.58,E2 -27167.58} C_VEL
LIN {X 0,Y 215.594,Z 843.615,A -85,B 0,C 180,E1 -27167.834,E2 -27167.834} C_VEL
LIN {X 0,Y 213.935,Z 839.27,A -85,B 0,C 180,E1 -27170.903,E2 -27170.903} C_VEL
LIN {X 0,Y 213.123,Z 837.079,A -85,B 0,C 180,E1 -27172.896,E2 -27172.896} C_VEL
LIN {X 0,Y 212.333,Z 834.688,A -85,B 0,C 180,E1 -27175.729,E2 -27175.729} C_VEL
LIN {X 0,Y 211.863,Z 833.253,A -85,B 0,C 180,E1 -27179.999,E2 -27179.999} C_VEL
LIN {X 0,Y 212.491,Z 835.068,A -85,B 0,C 180,E1 -27185.337,E2 -27185.337} C_VEL
LIN {X 0,Y 213.675,Z 838.483,A -85,B 0,C 180,E1 -27188.898,E2 -27188.898} C_VEL
LIN {X 0,Y 215.257,Z 842.668,A -85,B 0,C 180,E1 -27192.006,E2 -27192.006} C_VEL
LIN {X 0,Y 216.964,Z 847.496,A -85,B 0,C 180,E1 -27194.64,E2 -27194.64} C_VEL
LIN {X 0,Y 218.909,Z 853.334,A -85,B 0,C 180,E1 -27197.156,E2 -27197.156} C_VEL
LIN {X 0,Y 225.608,Z 870.041,A -85,B 0,C 180,E1 -27203.416,E2 -27203.416} C_VEL
LIN {X 0,Y 232.163,Z 881.112,A -85,B 0,C 180,E1 -27207.783,E2 -27207.783} C_VEL
LIN {X 0,Y 238.683,Z 889.893,A -85,B 0,C 180,E1 -27211.375,E2 -27211.375} C_VEL
LIN {X 0,Y 247.397,Z 899.547,A -85,B 0,C 180,E1 -27215.491,E2 -27215.491} C_VEL
LIN {X 0,Y 259.974,Z 911.355,A -85,B 0,C 180,E1 -27220.451,E2 -27220.451} C_VEL
LIN {X 0,Y 275.593,Z 923.661,A -85,B 0,C 180,E1 -27225.563,E2 -27225.563} C_VEL
LIN {X 0,Y 283.272,Z 929.693,A -85,B 0,C 180,E1 -27228.098,E2 -27228.098} C_VEL
LIN {X 0,Y 288.877,Z 933.964,A -85,B 0,C 180,E1 -27230.027,E2 -27230.027} C_VEL
LIN {X 0,Y 296.159,Z 939.464,A -85,B 0,C 180,E1 -27232.677,E2 -27232.677} C_VEL
LIN {X 0,Y 302.883,Z 944.849,A -85,B 0,C 180,E1 -27235.327,E2 -27235.327} C_VEL
LIN {X 0,Y 309.67,Z 949.791,A -85,B 0,C 180,E1 -27238.103,E2 -27238.103} C_VEL
LIN {X 0,Y 315.266,Z 954.146,A -85,B 0,C 180,E1 -27240.632,E2 -27240.632} C_VEL
LIN {X 0,Y 319.258,Z 956.869,A -85,B 0,C 180,E1 -27242.466,E2 -27242.466} C_VEL
LIN {X 0,Y 322.699,Z 959.36,A -85,B 0,C 180,E1 -27244.179,E2 -27244.179} C_VEL
LIN {X 0,Y 328.066,Z 963.359,A -85,B 0,C 180,E1 -27247.096,E2 -27247.096} C_VEL
LIN {X 0,Y 331.306,Z 965.451,A -85,B 0,C 180,E1 -27248.965,E2 -27248.965} C_VEL
LIN {X 0,Y 334.511,Z 967.487,A -85,B 0,C 180,E1 -27250.984,E2 -27250.984} C_VEL
LIN {X 0,Y 337.568,Z 970.037,A -85,B 0,C 180,E1 -27253.272,E2 -27253.272} C_VEL
LIN {X 0,Y 340.644,Z 972.308,A -85,B 0,C 180,E1 -27255.852,E2 -27255.852} C_VEL
LIN {X 0,Y 343.126,Z 973.814,A -85,B 0,C 180,E1 -27258.181,E2 -27258.181} C_VEL
LIN {X 0,Y 345.402,Z 974.827,A -85,B 0,C 180,E1 -27260.632,E2 -27260.632} C_VEL
LIN {X 0,Y 347.124,Z 975.611,A -85,B 0,C 180,E1 -27263.023,E2 -27263.023} C_VEL
LIN {X 0,Y 348.35,Z 976.189,A -85,B 0,C 180,E1 -27265.371,E2 -27265.371} C_VEL
LIN {X 0,Y 349.091,Z 976.493,A -85,B 0,C 180,E1 -27267.692,E2 -27267.692} C_VEL
LIN {X 0,Y 349.268,Z 976.643,A -85,B 0,C 180,E1 -27270,E2 -27270} C_VEL
LIN {X 0,Y 349.088,Z 976.49,A -85,B 0,C 180,E1 -27272.308,E2 -27272.308} C_VEL
LIN {X 0,Y 348.345,Z 976.203,A -85,B 0,C 180,E1 -27274.629,E2 -27274.629} C_VEL
LIN {X 0,Y 347.036,Z 975.58,A -85,B 0,C 180,E1 -27277.11,E2 -27277.11} C_VEL
LIN {X 0,Y 345.404,Z 974.812,A -85,B 0,C 180,E1 -27279.368,E2 -27279.368} C_VEL
LIN {X 0,Y 343.113,Z 973.837,A -85,B 0,C 180,E1 -27281.819,E2 -27281.819} C_VEL
LIN {X 0,Y 340.439,Z 972.169,A -85,B 0,C 180,E1 -27284.343,E2 -27284.343} C_VEL
LIN {X 0,Y 337.313,Z 969.766,A -85,B 0,C 180,E1 -27286.959,E2 -27286.959} C_VEL
LIN {X 0,Y 333.524,Z 966.687,A -85,B 0,C 180,E1 -27289.703,E2 -27289.703} C_VEL
LIN {X 0,Y 331.105,Z 965.314,A -85,B 0,C 180,E1 -27291.151,E2 -27291.151} C_VEL
LIN {X 0,Y 328.072,Z 963.341,A -85,B 0,C 180,E1 -27292.907,E2 -27292.907} C_VEL
LIN {X 0,Y 322.746,Z 959.316,A -85,B 0,C 180,E1 -27295.817,E2 -27295.817} C_VEL
LIN {X 0,Y 317.12,Z 955.414,A -85,B 0,C 180,E1 -27298.525,E2 -27298.525} C_VEL
LIN {X 0,Y 310.937,Z 950.864,A -85,B 0,C 180,E1 -27301.322,E2 -27301.322} C_VEL
LIN {X 0,Y 305.908,Z 947.041,A -85,B 0,C 180,E1 -27303.461,E2 -27303.461} C_VEL
LIN {X 0,Y 299.891,Z 942.499,A -85,B 0,C 180,E1 -27305.864,E2 -27305.864} C_VEL
LIN {X 0,Y 294.31,Z 938.095,A -85,B 0,C 180,E1 -27308,E2 -27308} C_VEL
LIN {X 0,Y 288.87,Z 933.934,A -85,B 0,C 180,E1 -27309.972,E2 -27309.972} C_VEL
LIN {X 0,Y 281.369,Z 928.227,A -85,B 0,C 180,E1 -27312.536,E2 -27312.536} C_VEL
LIN {X 0,Y 273.593,Z 922.109,A -85,B 0,C 180,E1 -27315.057,E2 -27315.057} C_VEL
LIN {X 0,Y 256.515,Z 908.252,A -85,B 0,C 180,E1 -27320.813,E2 -27320.813} C_VEL
LIN {X 0,Y 243.288,Z 895.333,A -85,B 0,C 180,E1 -27326.359,E2 -27326.359} C_VEL
LIN {X 0,Y 233.377,Z 882.885,A -85,B 0,C 180,E1 -27331.534,E2 -27331.534} C_VEL
LIN {X 0,Y 225.605,Z 870.052,A -85,B 0,C 180,E1 -27336.585,E2 -27336.585} C_VEL
LIN {X 0,Y 219.689,Z 855.71,A -85,B 0,C 180,E1 -27341.939,E2 -27341.939} C_VEL
LIN {X 0,Y 217.694,Z 849.601,A -85,B 0,C 180,E1 -27344.374,E2 -27344.374} C_VEL
LIN {X 0,Y 215.571,Z 843.54,A -85,B 0,C 180,E1 -27347.467,E2 -27347.467} C_VEL
LIN {X 0,Y 213.973,Z 839.326,A -85,B 0,C 180,E1 -27350.423,E2 -27350.423} C_VEL
LIN {X 0,Y 213.145,Z 837.16,A -85,B 0,C 180,E1 -27352.422,E2 -27352.422} C_VEL
LIN {X 0,Y 212.354,Z 834.676,A -85,B 0,C 180,E1 -27355.255,E2 -27355.255} C_VEL
LIN {X 0,Y 211.858,Z 833.295,A -85,B 0,C 180,E1 -27360.001,E2 -27360.001} C_VEL
LIN {X 0,Y 212.502,Z 835.124,A -85,B 0,C 180,E1 -27364.981,E2 -27364.981} C_VEL
LIN {X 0,Y 213.677,Z 838.567,A -85,B 0,C 180,E1 -27368.512,E2 -27368.512} C_VEL
LIN {X 0,Y 215.08,Z 842.273,A -85,B 0,C 180,E1 -27371.307,E2 -27371.307} C_VEL
LIN {X 0,Y 215.618,Z 843.642,A -85,B 0,C 180,E1 -27372.199,E2 -27372.199} C_VEL
LIN {X 0,Y 210.587,Z 887.484,A -85,B 0,C 180,E1 -27373.079,E2 -27373.079} C_VEL
LIN {X 0,Y 207.369,Z 904.368,A -85,B 0,C 180,E1 -27373.509,E2 -27373.509} C_VEL
LIN {X 0,Y 202.412,Z 921.941,A -85,B 0,C 180,E1 -27374.096,E2 -27374.096} C_VEL
LIN {X 0,Y 197.619,Z 935.196,A -85,B 0,C 180,E1 -27374.67,E2 -27374.67} C_VEL
LIN {X 0,Y 192.276,Z 947.678,A -85,B 0,C 180,E1 -27375.415,E2 -27375.415} C_VEL
LIN {X 0,Y 185.858,Z 960.405,A -85,B 0,C 180,E1 -27376.362,E2 -27376.362} C_VEL
LIN {X 0,Y 179.496,Z 971.39,A -85,B 0,C 180,E1 -27377.378,E2 -27377.378} C_VEL
LIN {X 0,Y 172.419,Z 982.179,A -85,B 0,C 180,E1 -27378.618,E2 -27378.618} C_VEL
LIN {X 0,Y 164.68,Z 992.668,A -85,B 0,C 180,E1 -27380.139,E2 -27380.139} C_VEL
LIN {X 0,Y 157.081,Z 1001.929,A -85,B 0,C 180,E1 -27381.82,E2 -27381.82} C_VEL
LIN {X 0,Y 148.132,Z 1011.651,A -85,B 0,C 180,E1 -27384.038,E2 -27384.038} C_VEL
LIN {X 0,Y 139.336,Z 1020.296,A -85,B 0,C 180,E1 -27386.618,E2 -27386.618} C_VEL
LIN {X 0,Y 129.827,Z 1028.766,A -85,B 0,C 180,E1 -27389.99,E2 -27389.99} C_VEL
LIN {X 0,Y 121.893,Z 1035.193,A -85,B 0,C 180,E1 -27393.279,E2 -27393.279} C_VEL
LIN {X 0,Y 111.887,Z 1042.619,A -85,B 0,C 180,E1 -27398.555,E2 -27398.555} C_VEL
LIN {X 0,Y 105.475,Z 1047.114,A -85,B 0,C 180,E1 -27402.867,E2 -27402.867} C_VEL
LIN {X 0,Y 97.72,Z 1052.224,A -85,B 0,C 180,E1 -27409.665,E2 -27409.665} C_VEL
LIN {X 0,Y 90.985,Z 1056.532,A -85,B 0,C 180,E1 -27418.178,E2 -27418.178} C_VEL
LIN {X 0,Y 86.979,Z 1059.22,A -85,B 0,C 180,E1 -27426.172,E2 -27426.172} C_VEL
LIN {X 0,Y 85.389,Z 1060.418,A -85,B 0,C 180,E1 -27430.779,E2 -27430.779} C_VEL
LIN {X 0,Y 83.806,Z 1061.918,A -85,B 0,C 180,E1 -27440.345,E2 -27440.345} C_VEL
LIN {X 0,Y 83.875,Z 1062.432,A -85,B 0,C 180,E1 -27450,E2 -27450} C_VEL
LIN {X 0,Y 83.806,Z 1061.918,A -85,B 0,C 180,E1 -27459.655,E2 -27459.655} C_VEL
LIN {X 0,Y 85.389,Z 1060.418,A -85,B 0,C 180,E1 -27469.221,E2 -27469.221} C_VEL
LIN {X 0,Y 88.999,Z 1057.926,A -85,B 0,C 180,E1 -27478.281,E2 -27478.281} C_VEL
LIN {X 0,Y 96.02,Z 1053.316,A -85,B 0,C 180,E1 -27488.471,E2 -27488.471} C_VEL
LIN {X 0,Y 101.429,Z 1049.816,A -85,B 0,C 180,E1 -27493.858,E2 -27493.858} C_VEL
LIN {X 0,Y 110.053,Z 1043.916,A -85,B 0,C 180,E1 -27500.311,E2 -27500.311} C_VEL
LIN {X 0,Y 116.899,Z 1039.017,A -85,B 0,C 180,E1 -27504.252,E2 -27504.252} C_VEL
LIN {X 0,Y 127.167,Z 1030.989,A -85,B 0,C 180,E1 -27508.937,E2 -27508.937} C_VEL
LIN {X 0,Y 135.869,Z 1023.441,A -85,B 0,C 180,E1 -27512.254,E2 -27512.254} C_VEL
LIN {X 0,Y 143.759,Z 1016.042,A -85,B 0,C 180,E1 -27514.741,E2 -27514.741} C_VEL
LIN {X 0,Y 152.517,Z 1006.935,A -85,B 0,C 180,E1 -27517.158,E2 -27517.158} C_VEL
LIN {X 0,Y 160.094,Z 998.38,A -85,B 0,C 180,E1 -27518.881,E2 -27518.881} C_VEL
LIN {X 0,Y 168.506,Z 987.645,A -85,B 0,C 180,E1 -27520.641,E2 -27520.641} C_VEL
LIN {X 0,Y 176.325,Z 976.371,A -85,B 0,C 180,E1 -27522.099,E2 -27522.099} C_VEL
LIN {X 0,Y 183.463,Z 964.715,A -85,B 0,C 180,E1 -27523.268,E2 -27523.268} C_VEL
LIN {X 0,Y 189.859,Z 952.701,A -85,B 0,C 180,E1 -27524.241,E2 -27524.241} C_VEL
LIN {X 0,Y 195.495,Z 940.391,A -85,B 0,C 180,E1 -27525.044,E2 -27525.044} C_VEL
LIN {X 0,Y 200.46,Z 927.643,A -85,B 0,C 180,E1 -27525.67,E2 -27525.67} C_VEL
LIN {X 0,Y 204.67,Z 914.439,A -85,B 0,C 180,E1 -27526.192,E2 -27526.192} C_VEL
LIN {X 0,Y 205.083,Z 912.964,A -85,B 0,C 180,E1 -27526.231,E2 -27526.231} C_VEL
LIN {X 0,Y 206.531,Z 907.34,A -85,B 0,C 180,E1 -27526.544,E2 -27526.544} C_VEL
LIN {X 0,Y 207.43,Z 901.849,A -85,B 0,C 180,E1 -27527.125,E2 -27527.125} C_VEL
LIN {X 0,Y 208.986,Z 889.062,A -85,B 0,C 180,E1 -27528.577,E2 -27528.577} C_VEL
LIN {X 0,Y 209.639,Z 883.3,A -85,B 0,C 180,E1 -27528.897,E2 -27528.897} C_VEL
LIN {X 0,Y 213.658,Z 848.47,A -85,B 0,C 180,E1 -27529.576,E2 -27529.576} C_VEL
LIN {X 0,Y 212.242,Z 844.316,A -85,B 0,C 180,E1 -27532.866,E2 -27532.866} C_VEL
LIN {X 0,Y 211.476,Z 841.797,A -85,B 0,C 180,E1 -27535.664,E2 -27535.664} C_VEL
LIN {X 0,Y 210.993,Z 840.344,A -85,B 0,C 180,E1 -27539.999,E2 -27539.999} C_VEL
LIN {X 0,Y 211.528,Z 842.015,A -85,B 0,C 180,E1 -27545.003,E2 -27545.003} C_VEL
LIN {X 0,Y 212.571,Z 845.321,A -85,B 0,C 180,E1 -27548.436,E2 -27548.436} C_VEL
LIN {X 0,Y 214.014,Z 849.394,A -85,B 0,C 180,E1 -27551.483,E2 -27551.483} C_VEL
LIN {X 0,Y 215.966,Z 855.459,A -85,B 0,C 180,E1 -27554.652,E2 -27554.652} C_VEL
LIN {X 0,Y 218.051,Z 862.312,A -85,B 0,C 180,E1 -27557.408,E2 -27557.408} C_VEL
LIN {X 0,Y 223.692,Z 876.52,A -85,B 0,C 180,E1 -27562.809,E2 -27562.809} C_VEL
LIN {X 0,Y 229.719,Z 887.24,A -85,B 0,C 180,E1 -27567.141,E2 -27567.141} C_VEL
LIN {X 0,Y 236.121,Z 896.367,A -85,B 0,C 180,E1 -27571.004,E2 -27571.004} C_VEL
LIN {X 0,Y 244.052,Z 905.534,A -85,B 0,C 180,E1 -27575.039,E2 -27575.039} C_VEL
LIN {X 0,Y 256.174,Z 917.206,A -85,B 0,C 180,E1 -27580.143,E2 -27580.143} C_VEL
LIN {X 0,Y 273.473,Z 930.99,A -85,B 0,C 180,E1 -27586.018,E2 -27586.018} C_VEL
LIN {X 0,Y 281.166,Z 936.878,A -85,B 0,C 180,E1 -27588.579,E2 -27588.579} C_VEL
LIN {X 0,Y 288.561,Z 942.718,A -85,B 0,C 180,E1 -27591.202,E2 -27591.202} C_VEL
LIN {X 0,Y 294.33,Z 947.037,A -85,B 0,C 180,E1 -27593.349,E2 -27593.349} C_VEL
LIN {X 0,Y 300.668,Z 952.004,A -85,B 0,C 180,E1 -27595.877,E2 -27595.877} C_VEL
LIN {X 0,Y 306.159,Z 955.975,A -85,B 0,C 180,E1 -27598.14,E2 -27598.14} C_VEL
LIN {X 0,Y 310.617,Z 959.511,A -85,B 0,C 180,E1 -27600.148,E2 -27600.148} C_VEL
LIN {X 0,Y 316.223,Z 963.382,A -85,B 0,C 180,E1 -27602.745,E2 -27602.745} C_VEL
LIN {X 0,Y 319.541,Z 965.817,A -85,B 0,C 180,E1 -27604.388,E2 -27604.388} C_VEL
LIN {X 0,Y 324.423,Z 969.417,A -85,B 0,C 180,E1 -27607.05,E2 -27607.05} C_VEL
LIN {X 0,Y 329.301,Z 972.478,A -85,B 0,C 180,E1 -27609.891,E2 -27609.891} C_VEL
LIN {X 0,Y 332.433,Z 974.838,A -85,B 0,C 180,E1 -27612.052,E2 -27612.052} C_VEL
LIN {X 0,Y 335.495,Z 977.314,A -85,B 0,C 180,E1 -27614.494,E2 -27614.494} C_VEL
LIN {X 0,Y 338.617,Z 979.398,A -85,B 0,C 180,E1 -27617.284,E2 -27617.284} C_VEL
LIN {X 0,Y 340.658,Z 980.495,A -85,B 0,C 180,E1 -27619.3,E2 -27619.3} C_VEL
LIN {X 0,Y 342.741,Z 981.395,A -85,B 0,C 180,E1 -27621.748,E2 -27621.748} C_VEL
LIN {X 0,Y 344.259,Z 982.039,A -85,B 0,C 180,E1 -27624.142,E2 -27624.142} C_VEL
LIN {X 0,Y 345.223,Z 982.55,A -85,B 0,C 180,E1 -27626.499,E2 -27626.499} C_VEL
LIN {X 0,Y 345.672,Z 982.762,A -85,B 0,C 180,E1 -27628.835,E2 -27628.835} C_VEL
LIN {X 0,Y 345.671,Z 982.759,A -85,B 0,C 180,E1 -27631.165,E2 -27631.165} C_VEL
LIN {X 0,Y 345.221,Z 982.56,A -85,B 0,C 180,E1 -27633.501,E2 -27633.501} C_VEL
LIN {X 0,Y 344.24,Z 982.076,A -85,B 0,C 180,E1 -27635.859,E2 -27635.859} C_VEL
LIN {X 0,Y 342.73,Z 981.409,A -85,B 0,C 180,E1 -27638.253,E2 -27638.253} C_VEL
LIN {X 0,Y 340.653,Z 980.501,A -85,B 0,C 180,E1 -27640.7,E2 -27640.7} C_VEL
LIN {X 0,Y 338.102,Z 979.071,A -85,B 0,C 180,E1 -27643.217,E2 -27643.217} C_VEL
LIN {X 0,Y 335.124,Z 977.055,A -85,B 0,C 180,E1 -27645.82,E2 -27645.82} C_VEL
LIN {X 0,Y 331.668,Z 974.168,A -85,B 0,C 180,E1 -27648.532,E2 -27648.532} C_VEL
LIN {X 0,Y 329.302,Z 972.467,A -85,B 0,C 180,E1 -27650.109,E2 -27650.109} C_VEL
LIN {X 0,Y 324.431,Z 969.404,A -85,B 0,C 180,E1 -27652.949,E2 -27652.949} C_VEL
LIN {X 0,Y 319.555,Z 965.763,A -85,B 0,C 180,E1 -27655.617,E2 -27655.617} C_VEL
LIN {X 0,Y 314.763,Z 962.304,A -85,B 0,C 180,E1 -27657.961,E2 -27657.961} C_VEL
LIN {X 0,Y 309.489,Z 958.65,A -85,B 0,C 180,E1 -27660.356,E2 -27660.356} C_VEL
LIN {X 0,Y 306.177,Z 956.018,A -85,B 0,C 180,E1 -27661.866,E2 -27661.866} C_VEL
LIN {X 0,Y 299.214,Z 950.892,A -85,B 0,C 180,E1 -27664.707,E2 -27664.707} C_VEL
LIN {X 0,Y 294.291,Z 947.017,A -85,B 0,C 180,E1 -27666.656,E2 -27666.656} C_VEL
LIN {X 0,Y 288.555,Z 942.628,A -85,B 0,C 180,E1 -27668.797,E2 -27668.797} C_VEL
LIN {X 0,Y 283.05,Z 938.293,A -85,B 0,C 180,E1 -27670.774,E2 -27670.774} C_VEL
LIN {X 0,Y 275.378,Z 932.555,A -85,B 0,C 180,E1 -27673.337,E2 -27673.337} C_VEL
LIN {X 0,Y 267.526,Z 926.401,A -85,B 0,C 180,E1 -27675.881,E2 -27675.881} C_VEL
LIN {X 0,Y 250.923,Z 912.375,A -85,B 0,C 180,E1 -27681.963,E2 -27681.963} C_VEL
LIN {X 0,Y 238.472,Z 899.352,A -85,B 0,C 180,E1 -27687.714,E2 -27687.714} C_VEL
LIN {X 0,Y 230.544,Z 888.597,A -85,B 0,C 180,E1 -27692.31,E2 -27692.31} C_VEL
LIN {X 0,Y 224.455,Z 878.021,A -85,B 0,C 180,E1 -27696.588,E2 -27696.588} C_VEL
LIN {X 0,Y 219.042,Z 865.38,A -85,B 0,C 180,E1 -27701.457,E2 -27701.457} C_VEL
LIN {X 0,Y 216.155,Z 856.022,A -85,B 0,C 180,E1 -27705.082,E2 -27705.082} C_VEL
LIN {X 0,Y 214.142,Z 849.771,A -85,B 0,C 180,E1 -27708.284,E2 -27708.284} C_VEL
LIN {X 0,Y 212.403,Z 844.688,A -85,B 0,C 180,E1 -27712.036,E2 -27712.036} C_VEL
LIN {X 0,Y 211.487,Z 841.765,A -85,B 0,C 180,E1 -27715.235,E2 -27715.235} C_VEL
LIN {X 0,Y 210.992,Z 840.354,A -85,B 0,C 180,E1 -27720.001,E2 -27720.001} C_VEL
LIN {X 0,Y 211.532,Z 841.983,A -85,B 0,C 180,E1 -27724.597,E2 -27724.597} C_VEL
LIN {X 0,Y 212.622,Z 845.503,A -85,B 0,C 180,E1 -27728.166,E2 -27728.166} C_VEL
LIN {X 0,Y 213.66,Z 848.458,A -85,B 0,C 180,E1 -27730.423,E2 -27730.423} C_VEL
LIN {X 0,Y 209.168,Z 886.816,A -85,B 0,C 180,E1 -27731.175,E2 -27731.175} C_VEL
LIN {X 0,Y 206.211,Z 902.302,A -85,B 0,C 180,E1 -27731.531,E2 -27731.531} C_VEL
LIN {X 0,Y 201.235,Z 920.48,A -85,B 0,C 180,E1 -27732.08,E2 -27732.08} C_VEL
LIN {X 0,Y 195.818,Z 935.285,A -85,B 0,C 180,E1 -27732.674,E2 -27732.674} C_VEL
LIN {X 0,Y 190.505,Z 947.472,A -85,B 0,C 180,E1 -27733.349,E2 -27733.349} C_VEL
LIN {X 0,Y 183.975,Z 960.198,A -85,B 0,C 180,E1 -27734.229,E2 -27734.229} C_VEL
LIN {X 0,Y 177.485,Z 971.183,A -85,B 0,C 180,E1 -27735.167,E2 -27735.167} C_VEL
LIN {X 0,Y 170.266,Z 981.972,A -85,B 0,C 180,E1 -27736.331,E2 -27736.331} C_VEL
LIN {X 0,Y 162.341,Z 992.459,A -85,B 0,C 180,E1 -27737.751,E2 -27737.751} C_VEL
LIN {X 0,Y 154.566,Z 1001.723,A -85,B 0,C 180,E1 -27739.359,E2 -27739.359} C_VEL
LIN {X 0,Y 145.353,Z 1011.443,A -85,B 0,C 180,E1 -27741.45,E2 -27741.45} C_VEL
LIN {X 0,Y 136.406,Z 1019.96,A -85,B 0,C 180,E1 -27743.865,E2 -27743.865} C_VEL
LIN {X 0,Y 126.366,Z 1028.557,A -85,B 0,C 180,E1 -27747.148,E2 -27747.148} C_VEL
LIN {X 0,Y 118.098,Z 1034.985,A -85,B 0,C 180,E1 -27750.36,E2 -27750.36} C_VEL
LIN {X 0,Y 107.792,Z 1042.248,A -85,B 0,C 180,E1 -27755.415,E2 -27755.415} C_VEL
LIN {X 0,Y 100.705,Z 1046.905,A -85,B 0,C 180,E1 -27759.857,E2 -27759.857} C_VEL
LIN {X 0,Y 92.338,Z 1052.015,A -85,B 0,C 180,E1 -27766.765,E2 -27766.765} C_VEL
LIN {X 0,Y 85.472,Z 1056.031,A -85,B 0,C 180,E1 -27774.861,E2 -27774.861} C_VEL
LIN {X 0,Y 80.471,Z 1059.012,A -85,B 0,C 180,E1 -27784.108,E2 -27784.108} C_VEL
LIN {X 0,Y 78.646,Z 1060.21,A -85,B 0,C 180,E1 -27789.057,E2 -27789.057} C_VEL
LIN {X 0,Y 76.757,Z 1061.71,A -85,B 0,C 180,E1 -27799.449,E2 -27799.449} C_VEL
LIN {X 0,Y 76.77,Z 1062.226,A -85,B 0,C 180,E1 -27810,E2 -27810} C_VEL
LIN {X 0,Y 76.757,Z 1061.71,A -85,B 0,C 180,E1 -27820.551,E2 -27820.551} C_VEL
LIN {X 0,Y 78.646,Z 1060.21,A -85,B 0,C 180,E1 -27830.943,E2 -27830.943} C_VEL
LIN {X 0,Y 82.72,Z 1057.717,A -85,B 0,C 180,E1 -27840.647,E2 -27840.647} C_VEL
LIN {X 0,Y 90.473,Z 1053.107,A -85,B 0,C 180,E1 -27851.32,E2 -27851.32} C_VEL
LIN {X 0,Y 96.365,Z 1049.608,A -85,B 0,C 180,E1 -27856.827,E2 -27856.827} C_VEL
LIN {X 0,Y 105.352,Z 1043.871,A -85,B 0,C 180,E1 -27863.177,E2 -27863.177} C_VEL
LIN {X 0,Y 112.845,Z 1038.809,A -85,B 0,C 180,E1 -27867.221,E2 -27867.221} C_VEL
LIN {X 0,Y 123.599,Z 1030.78,A -85,B 0,C 180,E1 -27871.802,E2 -27871.802} C_VEL
LIN {X 0,Y 132.042,Z 1023.797,A -85,B 0,C 180,E1 -27874.798,E2 -27874.798} C_VEL
LIN {X 0,Y 140.85,Z 1015.835,A -85,B 0,C 180,E1 -27877.379,E2 -27877.379} C_VEL
LIN {X 0,Y 149.879,Z 1006.728,A -85,B 0,C 180,E1 -27879.685,E2 -27879.685} C_VEL
LIN {X 0,Y 157.66,Z 998.173,A -85,B 0,C 180,E1 -27881.304,E2 -27881.304} C_VEL
LIN {X 0,Y 166.061,Z 987.733,A -85,B 0,C 180,E1 -27882.925,E2 -27882.925} C_VEL
LIN {X 0,Y 174.265,Z 976.165,A -85,B 0,C 180,E1 -27884.331,E2 -27884.331} C_VEL
LIN {X 0,Y 181.537,Z 964.509,A -85,B 0,C 180,E1 -27885.425,E2 -27885.425} C_VEL
LIN {X 0,Y 188.048,Z 952.494,A -85,B 0,C 180,E1 -27886.333,E2 -27886.333} C_VEL
LIN {X 0,Y 193.78,Z 940.185,A -85,B 0,C 180,E1 -27887.078,E2 -27887.078} C_VEL
LIN {X 0,Y 198.826,Z 927.42,A -85,B 0,C 180,E1 -27887.655,E2 -27887.655} C_VEL
LIN {X 0,Y 203.094,Z 914.234,A -85,B 0,C 180,E1 -27888.135,E2 -27888.135} C_VEL
LIN {X 0,Y 206.437,Z 901.326,A -85,B 0,C 180,E1 -27888.467,E2 -27888.467} C_VEL
LIN {X 0,Y 209.066,Z 887.239,A -85,B 0,C 180,E1 -27888.821,E2 -27888.821} C_VEL
LIN {X 0,Y 209.639,Z 883.3,A -85,B 0,C 180,E1 -27888.897,E2 -27888.897} C_VEL
LIN {X 0,Y 210.061,Z 879.452,A -85,B 0,C 180,E1 -27889.159,E2 -27889.159} C_VEL
LIN {X 0,Y 210.402,Z 867.608,A -85,B 0,C 180,E1 -27890.927,E2 -27890.927} C_VEL
LIN {X 0,Y 210.727,Z 863.745,A -85,B 0,C 180,E1 -27891.179,E2 -27891.179} C_VEL
LIN {X 0,Y 211.904,Z 853.448,A -85,B 0,C 180,E1 -27891.355,E2 -27891.355} C_VEL
LIN {X 0,Y 211.037,Z 850.744,A -85,B 0,C 180,E1 -27893.786,E2 -27893.786} C_VEL
LIN {X 0,Y 210.488,Z 848.691,A -85,B 0,C 180,E1 -27896.171,E2 -27896.171} C_VEL
LIN {X 0,Y 210.125,Z 847.41,A -85,B 0,C 180,E1 -27899.999,E2 -27899.999} C_VEL
LIN {X 0,Y 210.573,Z 848.947,A -85,B 0,C 180,E1 -27904.666,E2 -27904.666} C_VEL
LIN {X 0,Y 211.518,Z 852.256,A -85,B 0,C 180,E1 -27908.068,E2 -27908.068} C_VEL
LIN {X 0,Y 212.723,Z 855.95,A -85,B 0,C 180,E1 -27910.83,E2 -27910.83} C_VEL
LIN {X 0,Y 214.58,Z 862.199,A -85,B 0,C 180,E1 -27914.091,E2 -27914.091} C_VEL
LIN {X 0,Y 220.966,Z 881.463,A -85,B 0,C 180,E1 -27921.598,E2 -27921.598} C_VEL
LIN {X 0,Y 226.181,Z 891.819,A -85,B 0,C 180,E1 -27925.849,E2 -27925.849} C_VEL
LIN {X 0,Y 232.825,Z 902.057,A -85,B 0,C 180,E1 -27930.309,E2 -27930.309} C_VEL
LIN {X 0,Y 242.353,Z 913.354,A -85,B 0,C 180,E1 -27935.448,E2 -27935.448} C_VEL
LIN {X 0,Y 257.726,Z 927.525,A -85,B 0,C 180,E1 -27941.919,E2 -27941.919} C_VEL
LIN {X 0,Y 271.162,Z 938.18,A -85,B 0,C 180,E1 -27946.527,E2 -27946.527} C_VEL
LIN {X 0,Y 278.879,Z 944.01,A -85,B 0,C 180,E1 -27949.114,E2 -27949.114} C_VEL
LIN {X 0,Y 286.269,Z 949.791,A -85,B 0,C 180,E1 -27951.776,E2 -27951.776} C_VEL
LIN {X 0,Y 293.449,Z 955.394,A -85,B 0,C 180,E1 -27954.516,E2 -27954.516} C_VEL
LIN {X 0,Y 300.448,Z 960.538,A -85,B 0,C 180,E1 -27957.361,E2 -27957.361} C_VEL
LIN {X 0,Y 305.51,Z 964.528,A -85,B 0,C 180,E1 -27959.597,E2 -27959.597} C_VEL
LIN {X 0,Y 310.626,Z 968.167,A -85,B 0,C 180,E1 -27961.93,E2 -27961.93} C_VEL
LIN {X 0,Y 315.383,Z 971.524,A -85,B 0,C 180,E1 -27964.228,E2 -27964.228} C_VEL
LIN {X 0,Y 320.564,Z 975.365,A -85,B 0,C 180,E1 -27967.042,E2 -27967.042} C_VEL
LIN {X 0,Y 325.268,Z 978.314,A -85,B 0,C 180,E1 -27969.776,E2 -27969.776} C_VEL
LIN {X 0,Y 327.449,Z 979.877,A -85,B 0,C 180,E1 -27971.22,E2 -27971.22} C_VEL
LIN {X 0,Y 331.009,Z 982.781,A -85,B 0,C 180,E1 -27973.978,E2 -27973.978} C_VEL
LIN {X 0,Y 334.041,Z 984.92,A -85,B 0,C 180,E1 -27976.619,E2 -27976.619} C_VEL
LIN {X 0,Y 336.701,Z 986.39,A -85,B 0,C 180,E1 -27979.172,E2 -27979.172} C_VEL
LIN {X 0,Y 338.853,Z 987.327,A -85,B 0,C 180,E1 -27981.652,E2 -27981.652} C_VEL
LIN {X 0,Y 340.381,Z 987.98,A -85,B 0,C 180,E1 -27984.075,E2 -27984.075} C_VEL
LIN {X 0,Y 341.386,Z 988.489,A -85,B 0,C 180,E1 -27986.459,E2 -27986.459} C_VEL
LIN {X 0,Y 341.852,Z 988.718,A -85,B 0,C 180,E1 -27988.822,E2 -27988.822} C_VEL
LIN {X 0,Y 341.851,Z 988.714,A -85,B 0,C 180,E1 -27991.178,E2 -27991.178} C_VEL
LIN {X 0,Y 341.375,Z 988.513,A -85,B 0,C 180,E1 -27993.541,E2 -27993.541} C_VEL
LIN {X 0,Y 340.351,Z 988.023,A -85,B 0,C 180,E1 -27995.926,E2 -27995.926} C_VEL
LIN {X 0,Y 338.832,Z 987.355,A -85,B 0,C 180,E1 -27998.348,E2 -27998.348} C_VEL
LIN {X 0,Y 336.698,Z 986.397,A -85,B 0,C 180,E1 -28000.828,E2 -28000.828} C_VEL
LIN {X 0,Y 334.047,Z 984.909,A -85,B 0,C 180,E1 -28003.381,E2 -28003.381} C_VEL
LIN {X 0,Y 330.994,Z 982.8,A -85,B 0,C 180,E1 -28006.023,E2 -28006.023} C_VEL
LIN {X 0,Y 329.349,Z 981.404,A -85,B 0,C 180,E1 -28007.382,E2 -28007.382} C_VEL
LIN {X 0,Y 327.108,Z 979.593,A -85,B 0,C 180,E1 -28009.032,E2 -28009.032} C_VEL
LIN {X 0,Y 322.734,Z 976.765,A -85,B 0,C 180,E1 -28011.727,E2 -28011.727} C_VEL
LIN {X 0,Y 319.949,Z 974.933,A -85,B 0,C 180,E1 -28013.289,E2 -28013.289} C_VEL
LIN {X 0,Y 314.065,Z 970.458,A -85,B 0,C 180,E1 -28016.48,E2 -28016.48} C_VEL
LIN {X 0,Y 307.262,Z 965.788,A -85,B 0,C 180,E1 -28019.639,E2 -28019.639} C_VEL
LIN {X 0,Y 300.457,Z 960.555,A -85,B 0,C 180,E1 -28022.641,E2 -28022.641} C_VEL
LIN {X 0,Y 293.424,Z 955.337,A -85,B 0,C 180,E1 -28025.477,E2 -28025.477} C_VEL
LIN {X 0,Y 287.954,Z 951.003,A -85,B 0,C 180,E1 -28027.6,E2 -28027.6} C_VEL
LIN {X 0,Y 280.728,Z 945.495,A -85,B 0,C 180,E1 -28030.222,E2 -28030.222} C_VEL
LIN {X 0,Y 273.096,Z 939.703,A -85,B 0,C 180,E1 -28032.826,E2 -28032.826} C_VEL
LIN {X 0,Y 261.624,Z 930.742,A -85,B 0,C 180,E1 -28036.659,E2 -28036.659} C_VEL
LIN {X 0,Y 245.503,Z 916.691,A -85,B 0,C 180,E1 -28043.047,E2 -28043.047} C_VEL
LIN {X 0,Y 234.594,Z 904.381,A -85,B 0,C 180,E1 -28048.633,E2 -28048.633} C_VEL
LIN {X 0,Y 227.793,Z 894.596,A -85,B 0,C 180,E1 -28052.963,E2 -28052.963} C_VEL
LIN {X 0,Y 222.208,Z 884.043,A -85,B 0,C 180,E1 -28057.361,E2 -28057.361} C_VEL
LIN {X 0,Y 217.336,Z 871.811,A -85,B 0,C 180,E1 -28062.166,E2 -28062.166} C_VEL
LIN {X 0,Y 214.566,Z 862.17,A -85,B 0,C 180,E1 -28065.929,E2 -28065.929} C_VEL
LIN {X 0,Y 212.782,Z 856.136,A -85,B 0,C 180,E1 -28069.053,E2 -28069.053} C_VEL
LIN {X 0,Y 211.422,Z 851.877,A -85,B 0,C 180,E1 -28072.218,E2 -28072.218} C_VEL
LIN {X 0,Y 210.509,Z 848.669,A -85,B 0,C 180,E1 -28075.693,E2 -28075.693} C_VEL
LIN {X 0,Y 210.122,Z 847.437,A -85,B 0,C 180,E1 -28080.001,E2 -28080.001} C_VEL
LIN {X 0,Y 210.577,Z 849.028,A -85,B 0,C 180,E1 -28084.307,E2 -28084.307} C_VEL
LIN {X 0,Y 211.555,Z 852.356,A -85,B 0,C 180,E1 -28087.757,E2 -28087.757} C_VEL
LIN {X 0,Y 211.903,Z 853.458,A -85,B 0,C 180,E1 -28088.645,E2 -28088.645} C_VEL
LIN {X 0,Y 207.717,Z 887.822,A -85,B 0,C 180,E1 -28089.272,E2 -28089.272} C_VEL
LIN {X 0,Y 204.075,Z 905.824,A -85,B 0,C 180,E1 -28089.677,E2 -28089.677} C_VEL
LIN {X 0,Y 199.49,Z 921.349,A -85,B 0,C 180,E1 -28090.124,E2 -28090.124} C_VEL
LIN {X 0,Y 194.257,Z 935.382,A -85,B 0,C 180,E1 -28090.647,E2 -28090.647} C_VEL
LIN {X 0,Y 188.985,Z 947.266,A -85,B 0,C 180,E1 -28091.243,E2 -28091.243} C_VEL
LIN {X 0,Y 182.349,Z 959.991,A -85,B 0,C 180,E1 -28092.051,E2 -28092.051} C_VEL
LIN {X 0,Y 175.752,Z 970.976,A -85,B 0,C 180,E1 -28092.92,E2 -28092.92} C_VEL
LIN {X 0,Y 168.382,Z 981.763,A -85,B 0,C 180,E1 -28093.977,E2 -28093.977} C_VEL
LIN {X 0,Y 160.301,Z 992.252,A -85,B 0,C 180,E1 -28095.31,E2 -28095.31} C_VEL
LIN {X 0,Y 152.341,Z 1001.515,A -85,B 0,C 180,E1 -28096.816,E2 -28096.816} C_VEL
LIN {X 0,Y 142.877,Z 1011.235,A -85,B 0,C 180,E1 -28098.762,E2 -28098.762} C_VEL
LIN {X 0,Y 133.659,Z 1019.752,A -85,B 0,C 180,E1 -28101.045,E2 -28101.045} C_VEL
LIN {X 0,Y 123.23,Z 1028.347,A -85,B 0,C 180,E1 -28104.15,E2 -28104.15} C_VEL
LIN {X 0,Y 114.625,Z 1034.776,A -85,B 0,C 180,E1 -28107.251,E2 -28107.251} C_VEL
LIN {X 0,Y 103.785,Z 1042.04,A -85,B 0,C 180,E1 -28112.174,E2 -28112.174} C_VEL
LIN {X 0,Y 96.245,Z 1046.696,A -85,B 0,C 180,E1 -28116.561,E2 -28116.561} C_VEL
LIN {X 0,Y 87.213,Z 1051.806,A -85,B 0,C 180,E1 -28123.512,E2 -28123.512} C_VEL
LIN {X 0,Y 79.692,Z 1055.823,A -85,B 0,C 180,E1 -28131.88,E2 -28131.88} C_VEL
LIN {X 0,Y 74.054,Z 1058.804,A -85,B 0,C 180,E1 -28141.673,E2 -28141.673} C_VEL
LIN {X 0,Y 71.995,Z 1060.003,A -85,B 0,C 180,E1 -28147.017,E2 -28147.017} C_VEL
LIN {X 0,Y 69.743,Z 1061.504,A -85,B 0,C 180,E1 -28158.373,E2 -28158.373} C_VEL
LIN {X 0,Y 69.663,Z 1062.021,A -85,B 0,C 180,E1 -28170,E2 -28170} C_VEL
LIN {X 0,Y 69.743,Z 1061.504,A -85,B 0,C 180,E1 -28181.627,E2 -28181.627} C_VEL
LIN {X 0,Y 71.995,Z 1060.003,A -85,B 0,C 180,E1 -28192.983,E2 -28192.983} C_VEL
LIN {X 0,Y 78.34,Z 1056.537,A -85,B 0,C 180,E1 -28206.156,E2 -28206.156} C_VEL
LIN {X 0,Y 85.194,Z 1052.899,A -85,B 0,C 180,E1 -28214.522,E2 -28214.522} C_VEL
LIN {X 0,Y 91.571,Z 1049.399,A -85,B 0,C 180,E1 -28220.127,E2 -28220.127} C_VEL
LIN {X 0,Y 100.043,Z 1044.394,A -85,B 0,C 180,E1 -28225.805,E2 -28225.805} C_VEL
LIN {X 0,Y 109.102,Z 1038.6,A -85,B 0,C 180,E1 -28230.412,E2 -28230.412} C_VEL
LIN {X 0,Y 120.357,Z 1030.571,A -85,B 0,C 180,E1 -28234.832,E2 -28234.832} C_VEL
LIN {X 0,Y 129.144,Z 1023.589,A -85,B 0,C 180,E1 -28237.685,E2 -28237.685} C_VEL
LIN {X 0,Y 138.241,Z 1015.627,A -85,B 0,C 180,E1 -28240.134,E2 -28240.134} C_VEL
LIN {X 0,Y 147.542,Z 1006.52,A -85,B 0,C 180,E1 -28242.298,E2 -28242.298} C_VEL
LIN {X 0,Y 155.484,Z 998.004,A -85,B 0,C 180,E1 -28243.794,E2 -28243.794} C_VEL
LIN {X 0,Y 164.986,Z 986.33,A -85,B 0,C 180,E1 -28245.467,E2 -28245.467} C_VEL
LIN {X 0,Y 173.294,Z 974.713,A -85,B 0,C 180,E1 -28246.731,E2 -28246.731} C_VEL
LIN {X 0,Y 179.876,Z 964.302,A -85,B 0,C 180,E1 -28247.622,E2 -28247.622} C_VEL
LIN {X 0,Y 186.491,Z 952.288,A -85,B 0,C 180,E1 -28248.463,E2 -28248.463} C_VEL
LIN {X 0,Y 192.311,Z 939.978,A -85,B 0,C 180,E1 -28249.149,E2 -28249.149} C_VEL
LIN {X 0,Y 197.424,Z 927.213,A -85,B 0,C 180,E1 -28249.678,E2 -28249.678} C_VEL
LIN {X 0,Y 201.753,Z 914.029,A -85,B 0,C 180,E1 -28250.11,E2 -28250.11} C_VEL
LIN {X 0,Y 205.133,Z 901.12,A -85,B 0,C 180,E1 -28250.415,E2 -28250.415} C_VEL
LIN {X 0,Y 207.776,Z 887.263,A -85,B 0,C 180,E1 -28250.733,E2 -28250.733} C_VEL
LIN {X 0,Y 210.727,Z 863.745,A -85,B 0,C 180,E1 -28251.179,E2 -28251.179} C_VEL
LIN {X 0,Y 210.883,Z 861.192,A -85,B 0,C 180,E1 -28251.459,E2 -28251.459} C_VEL
LIN {X 0,Y 210.783,Z 858.854,A -85,B 0,C 180,E1 -28252.179,E2 -28252.179} C_VEL
LIN {X 0,Y 210.492,Z 857.279,A -85,B 0,C 180,E1 -28253.178,E2 -28253.178} C_VEL
LIN {X 0,Y 209.964,Z 856.189,A -85,B 0,C 180,E1 -28254.844,E2 -28254.844} C_VEL
LIN {X 0,Y 209.541,Z 855.642,A -85,B 0,C 180,E1 -28256.542,E2 -28256.542} C_VEL
LIN {X 0,Y 209.256,Z 854.492,A -85,B 0,C 180,E1 -28259.999,E2 -28259.999} C_VEL
LIN {X 0,Y 209.623,Z 855.909,A -85,B 0,C 180,E1 -28264.326,E2 -28264.326} C_VEL
LIN {X 0,Y 210.44,Z 859.044,A -85,B 0,C 180,E1 -28267.586,E2 -28267.586} C_VEL
LIN {X 0,Y 211.591,Z 862.96,A -85,B 0,C 180,E1 -28270.453,E2 -28270.453} C_VEL
LIN {X 0,Y 213.254,Z 869.207,A -85,B 0,C 180,E1 -28273.604,E2 -28273.604} C_VEL
LIN {X 0,Y 218.817,Z 887.556,A -85,B 0,C 180,E1 -28280.824,E2 -28280.824} C_VEL
LIN {X 0,Y 223.941,Z 898.705,A -85,B 0,C 180,E1 -28285.581,E2 -28285.581} C_VEL
LIN {X 0,Y 229.603,Z 907.977,A -85,B 0,C 180,E1 -28289.764,E2 -28289.764} C_VEL
LIN {X 0,Y 237.202,Z 917.505,A -85,B 0,C 180,E1 -28294.259,E2 -28294.259} C_VEL
LIN {X 0,Y 248.3,Z 928.748,A -85,B 0,C 180,E1 -28299.557,E2 -28299.557} C_VEL
LIN {X 0,Y 266.732,Z 943.697,A -85,B 0,C 180,E1 -28306.433,E2 -28306.433} C_VEL
LIN {X 0,Y 274.98,Z 949.972,A -85,B 0,C 180,E1 -28309.219,E2 -28309.219} C_VEL
LIN {X 0,Y 281.983,Z 955.439,A -85,B 0,C 180,E1 -28311.727,E2 -28311.727} C_VEL
LIN {X 0,Y 288.473,Z 960.508,A -85,B 0,C 180,E1 -28314.219,E2 -28314.219} C_VEL
LIN {X 0,Y 294.81,Z 965.226,A -85,B 0,C 180,E1 -28316.751,E2 -28316.751} C_VEL
LIN {X 0,Y 300.011,Z 969.165,A -85,B 0,C 180,E1 -28318.979,E2 -28318.979} C_VEL
LIN {X 0,Y 304.852,Z 972.782,A -85,B 0,C 180,E1 -28321.168,E2 -28321.168} C_VEL
LIN {X 0,Y 309.883,Z 976.227,A -85,B 0,C 180,E1 -28323.526,E2 -28323.526} C_VEL
LIN {X 0,Y 315.076,Z 980.217,A -85,B 0,C 180,E1 -28326.329,E2 -28326.329} C_VEL
LIN {X 0,Y 318.205,Z 982.314,A -85,B 0,C 180,E1 -28328.066,E2 -28328.066} C_VEL
LIN {X 0,Y 321.522,Z 984.337,A -85,B 0,C 180,E1 -28330.035,E2 -28330.035} C_VEL
LIN {X 0,Y 324.859,Z 986.911,A -85,B 0,C 180,E1 -28332.37,E2 -28332.37} C_VEL
LIN {X 0,Y 328.186,Z 989.512,A -85,B 0,C 180,E1 -28335.11,E2 -28335.11} C_VEL
LIN {X 0,Y 331.103,Z 991.406,A -85,B 0,C 180,E1 -28337.745,E2 -28337.745} C_VEL
LIN {X 0,Y 333.631,Z 992.628,A -85,B 0,C 180,E1 -28340.298,E2 -28340.298} C_VEL
LIN {X 0,Y 335.494,Z 993.422,A -85,B 0,C 180,E1 -28342.78,E2 -28342.78} C_VEL
LIN {X 0,Y 336.797,Z 994.034,A -85,B 0,C 180,E1 -28345.212,E2 -28345.212} C_VEL
LIN {X 0,Y 337.624,Z 994.394,A -85,B 0,C 180,E1 -28347.647,E2 -28347.647} C_VEL
LIN {X 0,Y 337.8,Z 994.54,A -85,B 0,C 180,E1 -28350,E2 -28350} C_VEL
LIN {X 0,Y 337.61,Z 994.387,A -85,B 0,C 180,E1 -28352.386,E2 -28352.386} C_VEL
LIN {X 0,Y 336.77,Z 994.071,A -85,B 0,C 180,E1 -28354.788,E2 -28354.788} C_VEL
LIN {X 0,Y 335.467,Z 993.452,A -85,B 0,C 180,E1 -28357.221,E2 -28357.221} C_VEL
LIN {X 0,Y 333.631,Z 992.625,A -85,B 0,C 180,E1 -28359.702,E2 -28359.702} C_VEL
LIN {X 0,Y 330.976,Z 991.347,A -85,B 0,C 180,E1 -28362.377,E2 -28362.377} C_VEL
LIN {X 0,Y 327.787,Z 989.24,A -85,B 0,C 180,E1 -28365.242,E2 -28365.242} C_VEL
LIN {X 0,Y 324.701,Z 986.775,A -85,B 0,C 180,E1 -28367.759,E2 -28367.759} C_VEL
LIN {X 0,Y 321.513,Z 984.354,A -85,B 0,C 180,E1 -28369.96,E2 -28369.96} C_VEL
LIN {X 0,Y 318.007,Z 982.124,A -85,B 0,C 180,E1 -28372.067,E2 -28372.067} C_VEL
LIN {X 0,Y 313.658,Z 979.128,A -85,B 0,C 180,E1 -28374.469,E2 -28374.469} C_VEL
LIN {X 0,Y 308.311,Z 975.05,A -85,B 0,C 180,E1 -28377.252,E2 -28377.252} C_VEL
LIN {X 0,Y 301.44,Z 970.317,A -85,B 0,C 180,E1 -28380.386,E2 -28380.386} C_VEL
LIN {X 0,Y 294.526,Z 965.02,A -85,B 0,C 180,E1 -28383.368,E2 -28383.368} C_VEL
LIN {X 0,Y 288.471,Z 960.476,A -85,B 0,C 180,E1 -28385.781,E2 -28385.781} C_VEL
LIN {X 0,Y 281.971,Z 955.365,A -85,B 0,C 180,E1 -28388.27,E2 -28388.27} C_VEL
LIN {X 0,Y 275.015,Z 949.977,A -85,B 0,C 180,E1 -28390.768,E2 -28390.768} C_VEL
LIN {X 0,Y 266.716,Z 943.745,A -85,B 0,C 180,E1 -28393.563,E2 -28393.563} C_VEL
LIN {X 0,Y 250.019,Z 930.224,A -85,B 0,C 180,E1 -28399.721,E2 -28399.721} C_VEL
LIN {X 0,Y 238.673,Z 919.228,A -85,B 0,C 180,E1 -28404.957,E2 -28404.957} C_VEL
LIN {X 0,Y 230.978,Z 909.816,A -85,B 0,C 180,E1 -28409.36,E2 -28409.36} C_VEL
LIN {X 0,Y 224.925,Z 900.544,A -85,B 0,C 180,E1 -28413.623,E2 -28413.623} C_VEL
LIN {X 0,Y 219.561,Z 889.38,A -85,B 0,C 180,E1 -28418.401,E2 -28418.401} C_VEL
LIN {X 0,Y 215.477,Z 877.789,A -85,B 0,C 180,E1 -28423.056,E2 -28423.056} C_VEL
LIN {X 0,Y 212.951,Z 868.018,A -85,B 0,C 180,E1 -28426.917,E2 -28426.917} C_VEL
LIN {X 0,Y 211.452,Z 862.452,A -85,B 0,C 180,E1 -28429.855,E2 -28429.855} C_VEL
LIN {X 0,Y 210.197,Z 858.076,A -85,B 0,C 180,E1 -28433.22,E2 -28433.22} C_VEL
LIN {X 0,Y 209.541,Z 855.6,A -85,B 0,C 180,E1 -28436.154,E2 -28436.154} C_VEL
LIN {X 0,Y 209.252,Z 854.521,A -85,B 0,C 180,E1 -28440.001,E2 -28440.001} C_VEL
LIN {X 0,Y 209.611,Z 855.844,A -85,B 0,C 180,E1 -28443.845,E2 -28443.845} C_VEL
LIN {X 0,Y 210.329,Z 858.655,A -85,B 0,C 180,E1 -28446.838,E2 -28446.838} C_VEL
LIN {X 0,Y 206.689,Z 887.655,A -85,B 0,C 180,E1 -28447.333,E2 -28447.333} C_VEL
LIN {X 0,Y 203.037,Z 905.501,A -85,B 0,C 180,E1 -28447.705,E2 -28447.705} C_VEL
LIN {X 0,Y 198.381,Z 921.096,A -85,B 0,C 180,E1 -28448.102,E2 -28448.102} C_VEL
LIN {X 0,Y 193.458,Z 934.286,A -85,B 0,C 180,E1 -28448.55,E2 -28448.55} C_VEL
LIN {X 0,Y 187.725,Z 947.059,A -85,B 0,C 180,E1 -28449.108,E2 -28449.108} C_VEL
LIN {X 0,Y 181.836,Z 958.349,A -85,B 0,C 180,E1 -28449.752,E2 -28449.752} C_VEL
LIN {X 0,Y 174.301,Z 970.771,A -85,B 0,C 180,E1 -28450.642,E2 -28450.642} C_VEL
LIN {X 0,Y 166.806,Z 981.557,A -85,B 0,C 180,E1 -28451.604,E2 -28451.604} C_VEL
LIN {X 0,Y 158.564,Z 992.045,A -85,B 0,C 180,E1 -28452.819,E2 -28452.819} C_VEL
LIN {X 0,Y 150.424,Z 1001.308,A -85,B 0,C 180,E1 -28454.201,E2 -28454.201} C_VEL
LIN {X 0,Y 140.737,Z 1011.027,A -85,B 0,C 180,E1 -28456,E2 -28456} C_VEL
LIN {X 0,Y 131.244,Z 1019.543,A -85,B 0,C 180,E1 -28458.108,E2 -28458.108} C_VEL
LIN {X 0,Y 120.462,Z 1028.139,A -85,B 0,C 180,E1 -28461.021,E2 -28461.021} C_VEL
LIN {X 0,Y 111.519,Z 1034.568,A -85,B 0,C 180,E1 -28463.968,E2 -28463.968} C_VEL
LIN {X 0,Y 100.135,Z 1041.832,A -85,B 0,C 180,E1 -28468.683,E2 -28468.683} C_VEL
LIN {X 0,Y 89.589,Z 1047.839,A -85,B 0,C 180,E1 -28474.545,E2 -28474.545} C_VEL
LIN {X 0,Y 82.411,Z 1051.597,A -85,B 0,C 180,E1 -28479.87,E2 -28479.87} C_VEL
LIN {X 0,Y 74.16,Z 1055.615,A -85,B 0,C 180,E1 -28488.443,E2 -28488.443} C_VEL
LIN {X 0,Y 67.798,Z 1058.595,A -85,B 0,C 180,E1 -28498.782,E2 -28498.782} C_VEL
LIN {X 0,Y 65.457,Z 1059.795,A -85,B 0,C 180,E1 -28504.567,E2 -28504.567} C_VEL
LIN {X 0,Y 62.77,Z 1061.297,A -85,B 0,C 180,E1 -28517.061,E2 -28517.061} C_VEL
LIN {X 0,Y 62.551,Z 1061.815,A -85,B 0,C 180,E1 -28530,E2 -28530} C_VEL
LIN {X 0,Y 62.77,Z 1061.297,A -85,B 0,C 180,E1 -28542.939,E2 -28542.939} C_VEL
LIN {X 0,Y 65.457,Z 1059.795,A -85,B 0,C 180,E1 -28555.433,E2 -28555.433} C_VEL
LIN {X 0,Y 72.132,Z 1056.577,A -85,B 0,C 180,E1 -28568.787,E2 -28568.787} C_VEL
LIN {X 0,Y 80.206,Z 1052.69,A -85,B 0,C 180,E1 -28578.141,E2 -28578.141} C_VEL
LIN {X 0,Y 87.125,Z 1049.19,A -85,B 0,C 180,E1 -28583.769,E2 -28583.769} C_VEL
LIN {X 0,Y 97.398,Z 1043.454,A -85,B 0,C 180,E1 -28589.982,E2 -28589.982} C_VEL
LIN {X 0,Y 105.73,Z 1038.391,A -85,B 0,C 180,E1 -28593.81,E2 -28593.81} C_VEL
LIN {X 0,Y 117.476,Z 1030.363,A -85,B 0,C 180,E1 -28598.012,E2 -28598.012} C_VEL
LIN {X 0,Y 126.583,Z 1023.38,A -85,B 0,C 180,E1 -28600.704,E2 -28600.704} C_VEL
LIN {X 0,Y 135.968,Z 1015.419,A -85,B 0,C 180,E1 -28602.982,E2 -28602.982} C_VEL
LIN {X 0,Y 145.528,Z 1006.313,A -85,B 0,C 180,E1 -28604.981,E2 -28604.981} C_VEL
LIN {X 0,Y 154.886,Z 996.336,A -85,B 0,C 180,E1 -28606.574,E2 -28606.574} C_VEL
LIN {X 0,Y 163.504,Z 985.906,A -85,B 0,C 180,E1 -28607.919,E2 -28607.919} C_VEL
LIN {X 0,Y 171.796,Z 974.506,A -85,B 0,C 180,E1 -28609.049,E2 -28609.049} C_VEL
LIN {X 0,Y 178.485,Z 964.096,A -85,B 0,C 180,E1 -28609.856,E2 -28609.856} C_VEL
LIN {X 0,Y 185.197,Z 952.081,A -85,B 0,C 180,E1 -28610.625,E2 -28610.625} C_VEL
LIN {X 0,Y 191.101,Z 939.773,A -85,B 0,C 180,E1 -28611.241,E2 -28611.241} C_VEL
LIN {X 0,Y 196.162,Z 927.326,A -85,B 0,C 180,E1 -28611.709,E2 -28611.709} C_VEL
LIN {X 0,Y 200.691,Z 913.703,A -85,B 0,C 180,E1 -28612.108,E2 -28612.108} C_VEL
LIN {X 0,Y 204.189,Z 900.346,A -85,B 0,C 180,E1 -28612.402,E2 -28612.402} C_VEL
LIN {X 0,Y 206.692,Z 887.457,A -85,B 0,C 180,E1 -28612.668,E2 -28612.668} C_VEL
LIN {X 0,Y 210.02,Z 861.297,A -85,B 0,C 180,E1 -28613.123,E2 -28613.123} C_VEL
LIN {X 0,Y 210.322,Z 858.623,A -85,B 0,C 180,E1 -28613.187,E2 -28613.187} C_VEL
LIN {X 0,Y 209.541,Z 855.642,A -85,B 0,C 180,E1 -28616.542,E2 -28616.542} C_VEL
LIN {X 0,Y 209.219,Z 855.863,A -85,B 0,C 180,E1 -28618.156,E2 -28618.156} C_VEL
LIN {X 0,Y 208.931,Z 857.179,A -85,B 0,C 180,E1 -28619.744,E2 -28619.744} C_VEL
LIN {X 0,Y 208.686,Z 862.672,A -85,B 0,C 180,E1 -28623.909,E2 -28623.909} C_VEL
LIN {X 0,Y 208.835,Z 863.799,A -85,B 0,C 180,E1 -28624.975,E2 -28624.975} C_VEL
LIN {X 0,Y 209.393,Z 865.947,A -85,B 0,C 180,E1 -28627.169,E2 -28627.169} C_VEL
LIN {X 0,Y 210.319,Z 869.415,A -85,B 0,C 180,E1 -28629.725,E2 -28629.725} C_VEL
LIN {X 0,Y 211.626,Z 874.887,A -85,B 0,C 180,E1 -28632.526,E2 -28632.526} C_VEL
LIN {X 0,Y 215.898,Z 891.93,A -85,B 0,C 180,E1 -28639.36,E2 -28639.36} C_VEL
LIN {X 0,Y 220.577,Z 903.684,A -85,B 0,C 180,E1 -28644.469,E2 -28644.469} C_VEL
LIN {X 0,Y 225.811,Z 913.174,A -85,B 0,C 180,E1 -28648.842,E2 -28648.842} C_VEL
LIN {X 0,Y 236.348,Z 926.595,A -85,B 0,C 180,E1 -28655.439,E2 -28655.439} C_VEL
LIN {X 0,Y 248.854,Z 938.453,A -85,B 0,C 180,E1 -28661.313,E2 -28661.313} C_VEL
LIN {X 0,Y 264.098,Z 950.609,A -85,B 0,C 180,E1 -28667.037,E2 -28667.037} C_VEL
LIN {X 0,Y 272.033,Z 956.676,A -85,B 0,C 180,E1 -28669.77,E2 -28669.77} C_VEL
LIN {X 0,Y 277.474,Z 960.894,A -85,B 0,C 180,E1 -28671.736,E2 -28671.736} C_VEL
LIN {X 0,Y 282.993,Z 965.166,A -85,B 0,C 180,E1 -28673.813,E2 -28673.813} C_VEL
LIN {X 0,Y 288.353,Z 969.348,A -85,B 0,C 180,E1 -28675.962,E2 -28675.962} C_VEL
LIN {X 0,Y 293.962,Z 973.402,A -85,B 0,C 180,E1 -28678.267,E2 -28678.267} C_VEL
LIN {X 0,Y 298.848,Z 977.235,A -85,B 0,C 180,E1 -28680.472,E2 -28680.472} C_VEL
LIN {X 0,Y 302.965,Z 980.089,A -85,B 0,C 180,E1 -28682.359,E2 -28682.359} C_VEL
LIN {X 0,Y 306.696,Z 982.757,A -85,B 0,C 180,E1 -28684.191,E2 -28684.191} C_VEL
LIN {X 0,Y 312.384,Z 986.924,A -85,B 0,C 180,E1 -28687.28,E2 -28687.28} C_VEL
LIN {X 0,Y 315.724,Z 989.058,A -85,B 0,C 180,E1 -28689.213,E2 -28689.213} C_VEL
LIN {X 0,Y 319.01,Z 991.331,A -85,B 0,C 180,E1 -28691.317,E2 -28691.317} C_VEL
LIN {X 0,Y 322.107,Z 993.844,A -85,B 0,C 180,E1 -28693.743,E2 -28693.743} C_VEL
LIN {X 0,Y 325.297,Z 996.088,A -85,B 0,C 180,E1 -28696.46,E2 -28696.46} C_VEL
LIN {X 0,Y 327.866,Z 997.562,A -85,B 0,C 180,E1 -28698.877,E2 -28698.877} C_VEL
LIN {X 0,Y 330.12,Z 998.587,A -85,B 0,C 180,E1 -28701.43,E2 -28701.43} C_VEL
LIN {X 0,Y 331.976,Z 999.392,A -85,B 0,C 180,E1 -28704.26,E2 -28704.26} C_VEL
LIN {X 0,Y 332.875,Z 999.849,A -85,B 0,C 180,E1 -28706.369,E2 -28706.369} C_VEL
LIN {X 0,Y 333.381,Z 1000.108,A -85,B 0,C 180,E1 -28708.792,E2 -28708.792} C_VEL
LIN {X 0,Y 333.38,Z 1000.105,A -85,B 0,C 180,E1 -28711.208,E2 -28711.208} C_VEL
LIN {X 0,Y 332.853,Z 999.879,A -85,B 0,C 180,E1 -28713.632,E2 -28713.632} C_VEL
LIN {X 0,Y 331.745,Z 999.344,A -85,B 0,C 180,E1 -28716.08,E2 -28716.08} C_VEL
LIN {X 0,Y 330.104,Z 998.601,A -85,B 0,C 180,E1 -28718.571,E2 -28718.571} C_VEL
LIN {X 0,Y 327.852,Z 997.582,A -85,B 0,C 180,E1 -28721.123,E2 -28721.123} C_VEL
LIN {X 0,Y 325.058,Z 995.929,A -85,B 0,C 180,E1 -28723.758,E2 -28723.758} C_VEL
LIN {X 0,Y 321.828,Z 993.605,A -85,B 0,C 180,E1 -28726.492,E2 -28726.492} C_VEL
LIN {X 0,Y 319.028,Z 991.279,A -85,B 0,C 180,E1 -28728.693,E2 -28728.693} C_VEL
LIN {X 0,Y 315.592,Z 988.963,A -85,B 0,C 180,E1 -28730.873,E2 -28730.873} C_VEL
LIN {X 0,Y 312.395,Z 986.895,A -85,B 0,C 180,E1 -28732.725,E2 -28732.725} C_VEL
LIN {X 0,Y 306.746,Z 982.715,A -85,B 0,C 180,E1 -28735.805,E2 -28735.805} C_VEL
LIN {X 0,Y 302.338,Z 979.583,A -85,B 0,C 180,E1 -28737.955,E2 -28737.955} C_VEL
LIN {X 0,Y 295.431,Z 974.641,A -85,B 0,C 180,E1 -28741.086,E2 -28741.086} C_VEL
LIN {X 0,Y 290.96,Z 971.197,A -85,B 0,C 180,E1 -28743.005,E2 -28743.005} C_VEL
LIN {X 0,Y 282.985,Z 965.176,A -85,B 0,C 180,E1 -28746.184,E2 -28746.184} C_VEL
LIN {X 0,Y 277.503,Z 960.878,A -85,B 0,C 180,E1 -28748.271,E2 -28748.271} C_VEL
LIN {X 0,Y 269.93,Z 955.021,A -85,B 0,C 180,E1 -28750.971,E2 -28750.971} C_VEL
LIN {X 0,Y 258.285,Z 946.06,A -85,B 0,C 180,E1 -28755.028,E2 -28755.028} C_VEL
LIN {X 0,Y 242.424,Z 932.722,A -85,B 0,C 180,E1 -28761.51,E2 -28761.51} C_VEL
LIN {X 0,Y 232.089,Z 921.756,A -85,B 0,C 180,E1 -28766.972,E2 -28766.972} C_VEL
LIN {X 0,Y 223.339,Z 909.145,A -85,B 0,C 180,E1 -28773.043,E2 -28773.043} C_VEL
LIN {X 0,Y 217.87,Z 897.5,A -85,B 0,C 180,E1 -28778.267,E2 -28778.267} C_VEL
LIN {X 0,Y 214.238,Z 886.235,A -85,B 0,C 180,E1 -28782.955,E2 -28782.955} C_VEL
LIN {X 0,Y 211.444,Z 874.09,A -85,B 0,C 180,E1 -28787.828,E2 -28787.828} C_VEL
LIN {X 0,Y 210.179,Z 868.877,A -85,B 0,C 180,E1 -28790.619,E2 -28790.619} C_VEL
LIN {X 0,Y 209.155,Z 864.837,A -85,B 0,C 180,E1 -28793.731,E2 -28793.731} C_VEL
LIN {X 0,Y 208.608,Z 862.564,A -85,B 0,C 180,E1 -28796.5,E2 -28796.5} C_VEL
LIN {X 0,Y 208.387,Z 861.565,A -85,B 0,C 180,E1 -28800.001,E2 -28800.001} C_VEL
LIN {X 0,Y 208.686,Z 862.907,A -85,B 0,C 180,E1 -28803.621,E2 -28803.621} C_VEL
LIN {X 0,Y 208.917,Z 864.123,A -85,B 0,C 180,E1 -28804.953,E2 -28804.953} C_VEL
LIN {X 0,Y 205.652,Z 889.014,A -85,B 0,C 180,E1 -28805.393,E2 -28805.393} C_VEL
LIN {X 0,Y 201.554,Z 907.558,A -85,B 0,C 180,E1 -28805.75,E2 -28805.75} C_VEL
LIN {X 0,Y 197.36,Z 921.296,A -85,B 0,C 180,E1 -28806.074,E2 -28806.074} C_VEL
LIN {X 0,Y 192.353,Z 934.485,A -85,B 0,C 180,E1 -28806.469,E2 -28806.469} C_VEL
LIN {X 0,Y 186.733,Z 946.854,A -85,B 0,C 180,E1 -28806.955,E2 -28806.955} C_VEL
LIN {X 0,Y 180.768,Z 958.143,A -85,B 0,C 180,E1 -28807.531,E2 -28807.531} C_VEL
LIN {X 0,Y 173.127,Z 970.564,A -85,B 0,C 180,E1 -28808.324,E2 -28808.324} C_VEL
LIN {X 0,Y 165.515,Z 981.35,A -85,B 0,C 180,E1 -28809.176,E2 -28809.176} C_VEL
LIN {X 0,Y 156.599,Z 992.442,A -85,B 0,C 180,E1 -28810.342,E2 -28810.342} C_VEL
LIN {X 0,Y 148.83,Z 1001.101,A -85,B 0,C 180,E1 -28811.529,E2 -28811.529} C_VEL
LIN {X 0,Y 138.933,Z 1010.82,A -85,B 0,C 180,E1 -28813.158,E2 -28813.158} C_VEL
LIN {X 0,Y 129.192,Z 1019.335,A -85,B 0,C 180,E1 -28815.08,E2 -28815.08} C_VEL
LIN {X 0,Y 118.074,Z 1027.931,A -85,B 0,C 180,E1 -28817.764,E2 -28817.764} C_VEL
LIN {X 0,Y 108.804,Z 1034.361,A -85,B 0,C 180,E1 -28820.515,E2 -28820.515} C_VEL
LIN {X 0,Y 96.873,Z 1041.622,A -85,B 0,C 180,E1 -28824.929,E2 -28824.929} C_VEL
LIN {X 0,Y 88.418,Z 1046.279,A -85,B 0,C 180,E1 -28829.035,E2 -28829.035} C_VEL
LIN {X 0,Y 77.979,Z 1051.388,A -85,B 0,C 180,E1 -28835.794,E2 -28835.794} C_VEL
LIN {X 0,Y 68.943,Z 1055.406,A -85,B 0,C 180,E1 -28844.475,E2 -28844.475} C_VEL
LIN {X 0,Y 61.749,Z 1058.387,A -85,B 0,C 180,E1 -28855.315,E2 -28855.315} C_VEL
LIN {X 0,Y 59.066,Z 1059.588,A -85,B 0,C 180,E1 -28861.58,E2 -28861.58} C_VEL
LIN {X 0,Y 55.817,Z 1061.09,A -85,B 0,C 180,E1 -28875.415,E2 -28875.415} C_VEL
LIN {X 0,Y 55.457,Z 1061.61,A -85,B 0,C 180,E1 -28890,E2 -28890} C_VEL
LIN {X 0,Y 55.817,Z 1061.09,A -85,B 0,C 180,E1 -28904.585,E2 -28904.585} C_VEL
LIN {X 0,Y 59.066,Z 1059.588,A -85,B 0,C 180,E1 -28918.42,E2 -28918.42} C_VEL
LIN {X 0,Y 66.195,Z 1056.584,A -85,B 0,C 180,E1 -28931.993,E2 -28931.993} C_VEL
LIN {X 0,Y 75.577,Z 1052.481,A -85,B 0,C 180,E1 -28942.223,E2 -28942.223} C_VEL
LIN {X 0,Y 83.067,Z 1048.981,A -85,B 0,C 180,E1 -28947.783,E2 -28947.783} C_VEL
LIN {X 0,Y 94.001,Z 1043.245,A -85,B 0,C 180,E1 -28953.786,E2 -28953.786} C_VEL
LIN {X 0,Y 102.76,Z 1038.183,A -85,B 0,C 180,E1 -28957.409,E2 -28957.409} C_VEL
LIN {X 0,Y 114.97,Z 1030.154,A -85,B 0,C 180,E1 -28961.346,E2 -28961.346} C_VEL
LIN {X 0,Y 124.393,Z 1023.172,A -85,B 0,C 180,E1 -28963.831,E2 -28963.831} C_VEL
LIN {X 0,Y 134.038,Z 1015.211,A -85,B 0,C 180,E1 -28965.927,E2 -28965.927} C_VEL
LIN {X 0,Y 143.844,Z 1006.107,A -85,B 0,C 180,E1 -28967.726,E2 -28967.726} C_VEL
LIN {X 0,Y 153.061,Z 996.494,A -85,B 0,C 180,E1 -28969.133,E2 -28969.133} C_VEL
LIN {X 0,Y 162.155,Z 985.698,A -85,B 0,C 180,E1 -28970.397,E2 -28970.397} C_VEL
LIN {X 0,Y 170.584,Z 974.3,A -85,B 0,C 180,E1 -28971.404,E2 -28971.404} C_VEL
LIN {X 0,Y 177.37,Z 963.89,A -85,B 0,C 180,E1 -28972.121,E2 -28972.121} C_VEL
LIN {X 0,Y 184.17,Z 951.875,A -85,B 0,C 180,E1 -28972.813,E2 -28972.813} C_VEL
LIN {X 0,Y 190.147,Z 939.567,A -85,B 0,C 180,E1 -28973.362,E2 -28973.362} C_VEL
LIN {X 0,Y 195.473,Z 926.534,A -85,B 0,C 180,E1 -28973.794,E2 -28973.794} C_VEL
LIN {X 0,Y 199.799,Z 913.636,A -85,B 0,C 180,E1 -28974.124,E2 -28974.124} C_VEL
LIN {X 0,Y 203.229,Z 900.786,A -85,B 0,C 180,E1 -28974.377,E2 -28974.377} C_VEL
LIN {X 0,Y 205.869,Z 887.491,A -85,B 0,C 180,E1 -28974.626,E2 -28974.626} C_VEL
LIN {X 0,Y 208.918,Z 864.107,A -85,B 0,C 180,E1 -28975.05,E2 -28975.05} C_VEL
LIN {X 0,Y 208.592,Z 862.573,A -85,B 0,C 180,E1 -28976.982,E2 -28976.982} C_VEL
LIN {X 0,Y 208.378,Z 861.645,A -85,B 0,C 180,E1 -28980.483,E2 -28980.483} C_VEL
LIN {X 0,Y 208.696,Z 862.973,A -85,B 0,C 180,E1 -28984.103,E2 -28984.103} C_VEL
LIN {X 0,Y 208.835,Z 863.799,A -85,B 0,C 180,E1 -28984.975,E2 -28984.975} C_VEL
LIN {X 0,Y 209.098,Z 865.999,A -85,B 0,C 180,E1 -28986.474,E2 -28986.474} C_VEL
LIN {X 0,Y 209.294,Z 869.311,A -85,B 0,C 180,E1 -28987.827,E2 -28987.827} C_VEL
LIN {X 0,Y 209.897,Z 879.803,A -85,B 0,C 180,E1 -28991.191,E2 -28991.191} C_VEL
LIN {X 0,Y 210.2,Z 882.062,A -85,B 0,C 180,E1 -28992.105,E2 -28992.105} C_VEL
LIN {X 0,Y 212.728,Z 895.104,A -85,B 0,C 180,E1 -28997.372,E2 -28997.372} C_VEL
LIN {X 0,Y 216.679,Z 907.55,A -85,B 0,C 180,E1 -29002.842,E2 -29002.842} C_VEL
LIN {X 0,Y 222.384,Z 919.001,A -85,B 0,C 180,E1 -29008.296,E2 -29008.296} C_VEL
LIN {X 0,Y 230.996,Z 930.674,A -85,B 0,C 180,E1 -29014.253,E2 -29014.253} C_VEL
LIN {X 0,Y 243.192,Z 942.88,A -85,B 0,C 180,E1 -29020.558,E2 -29020.558} C_VEL
LIN {X 0,Y 257.493,Z 954.466,A -85,B 0,C 180,E1 -29026.326,E2 -29026.326} C_VEL
LIN {X 0,Y 267.146,Z 961.829,A -85,B 0,C 180,E1 -29029.722,E2 -29029.722} C_VEL
LIN {X 0,Y 276.051,Z 968.716,A -85,B 0,C 180,E1 -29032.97,E2 -29032.97} C_VEL
LIN {X 0,Y 282.025,Z 973.418,A -85,B 0,C 180,E1 -29035.32,E2 -29035.32} C_VEL
LIN {X 0,Y 287.303,Z 977.256,A -85,B 0,C 180,E1 -29037.442,E2 -29037.442} C_VEL
LIN {X 0,Y 292.667,Z 981.473,A -85,B 0,C 180,E1 -29039.823,E2 -29039.823} C_VEL
LIN {X 0,Y 299.641,Z 986.378,A -85,B 0,C 180,E1 -29043.033,E2 -29043.033} C_VEL
LIN {X 0,Y 304.278,Z 989.808,A -85,B 0,C 180,E1 -29045.434,E2 -29045.434} C_VEL
LIN {X 0,Y 307.407,Z 992.052,A -85,B 0,C 180,E1 -29047.13,E2 -29047.13} C_VEL
LIN {X 0,Y 310.22,Z 993.887,A -85,B 0,C 180,E1 -29048.748,E2 -29048.748} C_VEL
LIN {X 0,Y 313.117,Z 995.759,A -85,B 0,C 180,E1 -29050.508,E2 -29050.508} C_VEL
LIN {X 0,Y 316.776,Z 998.662,A -85,B 0,C 180,E1 -29053.237,E2 -29053.237} C_VEL
LIN {X 0,Y 320.127,Z 1001.092,A -85,B 0,C 180,E1 -29056.026,E2 -29056.026} C_VEL
LIN {X 0,Y 322.995,Z 1002.786,A -85,B 0,C 180,E1 -29058.707,E2 -29058.707} C_VEL
LIN {X 0,Y 325.344,Z 1003.891,A -85,B 0,C 180,E1 -29061.303,E2 -29061.303} C_VEL
LIN {X 0,Y 327.078,Z 1004.658,A -85,B 0,C 180,E1 -29063.833,E2 -29063.833} C_VEL
LIN {X 0,Y 328.239,Z 1005.212,A -85,B 0,C 180,E1 -29066.317,E2 -29066.317} C_VEL
LIN {X 0,Y 328.76,Z 1005.497,A -85,B 0,C 180,E1 -29068.775,E2 -29068.775} C_VEL
LIN {X 0,Y 328.759,Z 1005.493,A -85,B 0,C 180,E1 -29071.225,E2 -29071.225} C_VEL
LIN {X 0,Y 328.613,Z 1005.367,A -85,B 0,C 180,E1 -29072.451,E2 -29072.451} C_VEL
LIN {X 0,Y 327.693,Z 1004.999,A -85,B 0,C 180,E1 -29074.921,E2 -29074.921} C_VEL
LIN {X 0,Y 326.14,Z 1004.272,A -85,B 0,C 180,E1 -29077.589,E2 -29077.589} C_VEL
LIN {X 0,Y 324.241,Z 1003.41,A -85,B 0,C 180,E1 -29079.985,E2 -29079.985} C_VEL
LIN {X 0,Y 321.633,Z 1002.041,A -85,B 0,C 180,E1 -29082.621,E2 -29082.621} C_VEL
LIN {X 0,Y 318.49,Z 999.98,A -85,B 0,C 180,E1 -29085.355,E2 -29085.355} C_VEL
LIN {X 0,Y 314.964,Z 997.138,A -85,B 0,C 180,E1 -29088.203,E2 -29088.203} C_VEL
LIN {X 0,Y 312.811,Z 995.539,A -85,B 0,C 180,E1 -29089.694,E2 -29089.694} C_VEL
LIN {X 0,Y 309.758,Z 993.569,A -85,B 0,C 180,E1 -29091.53,E2 -29091.53} C_VEL
LIN {X 0,Y 306.379,Z 991.327,A -85,B 0,C 180,E1 -29093.43,E2 -29093.43} C_VEL
LIN {X 0,Y 301.02,Z 987.24,A -85,B 0,C 180,E1 -29096.333,E2 -29096.333} C_VEL
LIN {X 0,Y 294.558,Z 982.784,A -85,B 0,C 180,E1 -29099.341,E2 -29099.341} C_VEL
LIN {X 0,Y 289.213,Z 978.707,A -85,B 0,C 180,E1 -29101.734,E2 -29101.734} C_VEL
LIN {X 0,Y 282.017,Z 973.374,A -85,B 0,C 180,E1 -29104.678,E2 -29104.678} C_VEL
LIN {X 0,Y 276.011,Z 968.679,A -85,B 0,C 180,E1 -29107.032,E2 -29107.032} C_VEL
LIN {X 0,Y 269.314,Z 963.529,A -85,B 0,C 180,E1 -29109.493,E2 -29109.493} C_VEL
LIN {X 0,Y 261.655,Z 957.665,A -85,B 0,C 180,E1 -29112.181,E2 -29112.181} C_VEL
LIN {X 0,Y 248.334,Z 947.282,A -85,B 0,C 180,E1 -29117.219,E2 -29117.219} C_VEL
LIN {X 0,Y 233.099,Z 933.168,A -85,B 0,C 180,E1 -29124.492,E2 -29124.492} C_VEL
LIN {X 0,Y 224.65,Z 922.418,A -85,B 0,C 180,E1 -29129.965,E2 -29129.965} C_VEL
LIN {X 0,Y 218.743,Z 912.169,A -85,B 0,C 180,E1 -29134.996,E2 -29134.996} C_VEL
LIN {X 0,Y 214.612,Z 901.566,A -85,B 0,C 180,E1 -29139.827,E2 -29139.827} C_VEL
LIN {X 0,Y 211.496,Z 889.252,A -85,B 0,C 180,E1 -29145.038,E2 -29145.038} C_VEL
LIN {X 0,Y 209.866,Z 879.97,A -85,B 0,C 180,E1 -29148.837,E2 -29148.837} C_VEL
LIN {X 0,Y 208.93,Z 875.236,A -85,B 0,C 180,E1 -29151.43,E2 -29151.43} C_VEL
LIN {X 0,Y 208.094,Z 871.546,A -85,B 0,C 180,E1 -29154.368,E2 -29154.368} C_VEL
LIN {X 0,Y 207.683,Z 869.528,A -85,B 0,C 180,E1 -29156.848,E2 -29156.848} C_VEL
LIN {X 0,Y 207.518,Z 868.642,A -85,B 0,C 180,E1 -29160.001,E2 -29160.001} C_VEL
LIN {X 0,Y 207.736,Z 869.699,A -85,B 0,C 180,E1 -29163.115,E2 -29163.115} C_VEL
LIN {X 0,Y 204.618,Z 891.678,A -85,B 0,C 180,E1 -29163.458,E2 -29163.458} C_VEL
LIN {X 0,Y 200.669,Z 908.38,A -85,B 0,C 180,E1 -29163.755,E2 -29163.755} C_VEL
LIN {X 0,Y 196.668,Z 921.279,A -85,B 0,C 180,E1 -29164.023,E2 -29164.023} C_VEL
LIN {X 0,Y 191.876,Z 933.839,A -85,B 0,C 180,E1 -29164.347,E2 -29164.347} C_VEL
LIN {X 0,Y 186.005,Z 946.648,A -85,B 0,C 180,E1 -29164.779,E2 -29164.779} C_VEL
LIN {X 0,Y 179.111,Z 959.373,A -85,B 0,C 180,E1 -29165.352,E2 -29165.352} C_VEL
LIN {X 0,Y 172.239,Z 970.358,A -85,B 0,C 180,E1 -29165.978,E2 -29165.978} C_VEL
LIN {X 0,Y 164.529,Z 981.144,A -85,B 0,C 180,E1 -29166.726,E2 -29166.726} C_VEL
LIN {X 0,Y 156.014,Z 991.631,A -85,B 0,C 180,E1 -29167.688,E2 -29167.688} C_VEL
LIN {X 0,Y 147.567,Z 1000.894,A -85,B 0,C 180,E1 -29168.808,E2 -29168.808} C_VEL
LIN {X 0,Y 137.472,Z 1010.612,A -85,B 0,C 180,E1 -29170.233,E2 -29170.233} C_VEL
LIN {X 0,Y 127.512,Z 1019.128,A -85,B 0,C 180,E1 -29171.962,E2 -29171.962} C_VEL
LIN {X 0,Y 116.086,Z 1027.723,A -85,B 0,C 180,E1 -29174.388,E2 -29174.388} C_VEL
LIN {X 0,Y 106.494,Z 1034.153,A -85,B 0,C 180,E1 -29176.884,E2 -29176.884} C_VEL
LIN {X 0,Y 94.058,Z 1041.414,A -85,B 0,C 180,E1 -29180.937,E2 -29180.937} C_VEL
LIN {X 0,Y 85.145,Z 1046.07,A -85,B 0,C 180,E1 -29184.779,E2 -29184.779} C_VEL
LIN {X 0,Y 73.989,Z 1051.179,A -85,B 0,C 180,E1 -29191.255,E2 -29191.255} C_VEL
LIN {X 0,Y 64.095,Z 1055.198,A -85,B 0,C 180,E1 -29199.868,E2 -29199.868} C_VEL
LIN {X 0,Y 55.981,Z 1058.178,A -85,B 0,C 180,E1 -29211.119,E2 -29211.119} C_VEL
LIN {X 0,Y 52.851,Z 1059.38,A -85,B 0,C 180,E1 -29217.866,E2 -29217.866} C_VEL
LIN {X 0,Y 48.931,Z 1060.883,A -85,B 0,C 180,E1 -29233.306,E2 -29233.306} C_VEL
LIN {X 0,Y 48.347,Z 1061.404,A -85,B 0,C 180,E1 -29250,E2 -29250} C_VEL
LIN {X 0,Y 48.931,Z 1060.883,A -85,B 0,C 180,E1 -29266.694,E2 -29266.694} C_VEL
LIN {X 0,Y 52.851,Z 1059.38,A -85,B 0,C 180,E1 -29282.134,E2 -29282.134} C_VEL
LIN {X 0,Y 60.506,Z 1056.591,A -85,B 0,C 180,E1 -29295.818,E2 -29295.818} C_VEL
LIN {X 0,Y 71.389,Z 1052.272,A -85,B 0,C 180,E1 -29306.8,E2 -29306.8} C_VEL
LIN {X 0,Y 79.451,Z 1048.772,A -85,B 0,C 180,E1 -29312.196,E2 -29312.196} C_VEL
LIN {X 0,Y 88.611,Z 1044.356,A -85,B 0,C 180,E1 -29316.85,E2 -29316.85} C_VEL
LIN {X 0,Y 100.213,Z 1037.975,A -85,B 0,C 180,E1 -29321.215,E2 -29321.215} C_VEL
LIN {X 0,Y 112.87,Z 1029.945,A -85,B 0,C 180,E1 -29324.819,E2 -29324.819} C_VEL
LIN {X 0,Y 122.591,Z 1022.965,A -85,B 0,C 180,E1 -29327.049,E2 -29327.049} C_VEL
LIN {X 0,Y 132.469,Z 1015.002,A -85,B 0,C 180,E1 -29328.953,E2 -29328.953} C_VEL
LIN {X 0,Y 142.499,Z 1005.901,A -85,B 0,C 180,E1 -29330.528,E2 -29330.528} C_VEL
LIN {X 0,Y 151.538,Z 996.665,A -85,B 0,C 180,E1 -29331.744,E2 -29331.744} C_VEL
LIN {X 0,Y 161.114,Z 985.491,A -85,B 0,C 180,E1 -29332.911,E2 -29332.911} C_VEL
LIN {X 0,Y 169.66,Z 974.092,A -85,B 0,C 180,E1 -29333.799,E2 -29333.799} C_VEL
LIN {X 0,Y 177.393,Z 962.247,A -85,B 0,C 180,E1 -29334.49,E2 -29334.49} C_VEL
LIN {X 0,Y 183.415,Z 951.669,A -85,B 0,C 180,E1 -29335.023,E2 -29335.023} C_VEL
LIN {X 0,Y 189.456,Z 939.361,A -85,B 0,C 180,E1 -29335.5,E2 -29335.5} C_VEL
LIN {X 0,Y 194.645,Z 926.848,A -85,B 0,C 180,E1 -29335.858,E2 -29335.858} C_VEL
LIN {X 0,Y 199.27,Z 913.185,A -85,B 0,C 180,E1 -29336.16,E2 -29336.16} C_VEL
LIN {X 0,Y 202.496,Z 901.32,A -85,B 0,C 180,E1 -29336.36,E2 -29336.36} C_VEL
LIN {X 0,Y 205.354,Z 887.105,A -85,B 0,C 180,E1 -29336.599,E2 -29336.599} C_VEL
LIN {X 0,Y 207.741,Z 869.663,A -85,B 0,C 180,E1 -29336.881,E2 -29336.881} C_VEL
LIN {X 0,Y 207.511,Z 868.708,A -85,B 0,C 180,E1 -29340.485,E2 -29340.485} C_VEL
LIN {X 0,Y 207.753,Z 869.859,A -85,B 0,C 180,E1 -29343.697,E2 -29343.697} C_VEL
LIN {X 0,Y 208.336,Z 872.727,A -85,B 0,C 180,E1 -29346.658,E2 -29346.658} C_VEL
LIN {X 0,Y 209.067,Z 875.786,A -85,B 0,C 180,E1 -29348.944,E2 -29348.944} C_VEL
LIN {X 0,Y 210.142,Z 881.646,A -85,B 0,C 180,E1 -29351.942,E2 -29351.942} C_VEL
LIN {X 0,Y 210.2,Z 882.062,A -85,B 0,C 180,E1 -29352.105,E2 -29352.105} C_VEL
LIN {X 0,Y 210.439,Z 884.666,A -85,B 0,C 180,E1 -29352.916,E2 -29352.916} C_VEL
LIN {X 0,Y 210.294,Z 890.336,A -85,B 0,C 180,E1 -29353.9,E2 -29353.9} C_VEL
LIN {X 0,Y 209.889,Z 896.138,A -85,B 0,C 180,E1 -29354.864,E2 -29354.864} C_VEL
LIN {X 0,Y 209.985,Z 898.945,A -85,B 0,C 180,E1 -29355.647,E2 -29355.647} C_VEL
LIN {X 0,Y 212.979,Z 911.335,A -85,B 0,C 180,E1 -29361.156,E2 -29361.156} C_VEL
LIN {X 0,Y 218.411,Z 924.016,A -85,B 0,C 180,E1 -29367.338,E2 -29367.338} C_VEL
LIN {X 0,Y 226.961,Z 936.317,A -85,B 0,C 180,E1 -29373.874,E2 -29373.874} C_VEL
LIN {X 0,Y 237.132,Z 946.981,A -85,B 0,C 180,E1 -29379.596,E2 -29379.596} C_VEL
LIN {X 0,Y 252.738,Z 959.738,A -85,B 0,C 180,E1 -29386.301,E2 -29386.301} C_VEL
LIN {X 0,Y 263.272,Z 967.794,A -85,B 0,C 180,E1 -29390.159,E2 -29390.159} C_VEL
LIN {X 0,Y 270.073,Z 972.95,A -85,B 0,C 180,E1 -29392.621,E2 -29392.621} C_VEL
LIN {X 0,Y 276.721,Z 978.221,A -85,B 0,C 180,E1 -29395.24,E2 -29395.24} C_VEL
LIN {X 0,Y 282.763,Z 982.628,A -85,B 0,C 180,E1 -29397.677,E2 -29397.677} C_VEL
LIN {X 0,Y 286.339,Z 985.42,A -85,B 0,C 180,E1 -29399.209,E2 -29399.209} C_VEL
LIN {X 0,Y 293.336,Z 990.551,A -85,B 0,C 180,E1 -29402.432,E2 -29402.432} C_VEL
LIN {X 0,Y 298.296,Z 994.121,A -85,B 0,C 180,E1 -29404.908,E2 -29404.908} C_VEL
LIN {X 0,Y 301.555,Z 996.526,A -85,B 0,C 180,E1 -29406.66,E2 -29406.66} C_VEL
LIN {X 0,Y 304.525,Z 998.494,A -85,B 0,C 180,E1 -29408.331,E2 -29408.331} C_VEL
LIN {X 0,Y 307.218,Z 1000.255,A -85,B 0,C 180,E1 -29409.932,E2 -29409.932} C_VEL
LIN {X 0,Y 310.289,Z 1002.504,A -85,B 0,C 180,E1 -29412.042,E2 -29412.042} C_VEL
LIN {X 0,Y 313.478,Z 1004.99,A -85,B 0,C 180,E1 -29414.585,E2 -29414.585} C_VEL
LIN {X 0,Y 316.426,Z 1006.989,A -85,B 0,C 180,E1 -29417.168,E2 -29417.168} C_VEL
LIN {X 0,Y 319.149,Z 1008.441,A -85,B 0,C 180,E1 -29419.854,E2 -29419.854} C_VEL
LIN {X 0,Y 321.299,Z 1009.397,A -85,B 0,C 180,E1 -29422.459,E2 -29422.459} C_VEL
LIN {X 0,Y 322.811,Z 1010.092,A -85,B 0,C 180,E1 -29425.004,E2 -29425.004} C_VEL
LIN {X 0,Y 323.718,Z 1010.498,A -85,B 0,C 180,E1 -29427.511,E2 -29427.511} C_VEL
LIN {X 0,Y 323.933,Z 1010.635,A -85,B 0,C 180,E1 -29430,E2 -29430} C_VEL
LIN {X 0,Y 323.641,Z 1010.473,A -85,B 0,C 180,E1 -29432.692,E2 -29432.692} C_VEL
LIN {X 0,Y 322.77,Z 1010.135,A -85,B 0,C 180,E1 -29434.996,E2 -29434.996} C_VEL
LIN {X 0,Y 321.274,Z 1009.419,A -85,B 0,C 180,E1 -29437.542,E2 -29437.542} C_VEL
LIN {X 0,Y 319.146,Z 1008.445,A -85,B 0,C 180,E1 -29440.146,E2 -29440.146} C_VEL
LIN {X 0,Y 316.445,Z 1006.972,A -85,B 0,C 180,E1 -29442.832,E2 -29442.832} C_VEL
LIN {X 0,Y 313.209,Z 1004.831,A -85,B 0,C 180,E1 -29445.62,E2 -29445.62} C_VEL
LIN {X 0,Y 309.535,Z 1001.868,A -85,B 0,C 180,E1 -29448.534,E2 -29448.534} C_VEL
LIN {X 0,Y 307.016,Z 1000.129,A -85,B 0,C 180,E1 -29450.193,E2 -29450.193} C_VEL
LIN {X 0,Y 303.605,Z 997.877,A -85,B 0,C 180,E1 -29452.191,E2 -29452.191} C_VEL
LIN {X 0,Y 300.208,Z 995.52,A -85,B 0,C 180,E1 -29454.078,E2 -29454.078} C_VEL
LIN {X 0,Y 294.771,Z 991.427,A -85,B 0,C 180,E1 -29456.936,E2 -29456.936} C_VEL
LIN {X 0,Y 289.847,Z 988.04,A -85,B 0,C 180,E1 -29459.204,E2 -29459.204} C_VEL
LIN {X 0,Y 282.776,Z 982.661,A -85,B 0,C 180,E1 -29462.327,E2 -29462.327} C_VEL
LIN {X 0,Y 275.463,Z 977.211,A -85,B 0,C 180,E1 -29465.272,E2 -29465.272} C_VEL
LIN {X 0,Y 270.143,Z 973.029,A -85,B 0,C 180,E1 -29467.343,E2 -29467.343} C_VEL
LIN {X 0,Y 262.293,Z 966.976,A -85,B 0,C 180,E1 -29470.213,E2 -29470.213} C_VEL
LIN {X 0,Y 247.269,Z 955.425,A -85,B 0,C 180,E1 -29475.866,E2 -29475.866} C_VEL
LIN {X 0,Y 232.525,Z 942.465,A -85,B 0,C 180,E1 -29482.809,E2 -29482.809} C_VEL
LIN {X 0,Y 222.07,Z 929.898,A -85,B 0,C 180,E1 -29489.579,E2 -29489.579} C_VEL
LIN {X 0,Y 216.094,Z 919.337,A -85,B 0,C 180,E1 -29494.989,E2 -29494.989} C_VEL
LIN {X 0,Y 212.197,Z 908.718,A -85,B 0,C 180,E1 -29500.029,E2 -29500.029} C_VEL
LIN {X 0,Y 209.853,Z 898.234,A -85,B 0,C 180,E1 -29504.652,E2 -29504.652} C_VEL
LIN {X 0,Y 208.317,Z 886.136,A -85,B 0,C 180,E1 -29509.701,E2 -29509.701} C_VEL
LIN {X 0,Y 207.62,Z 881.602,A -85,B 0,C 180,E1 -29512.219,E2 -29512.219} C_VEL
LIN {X 0,Y 207.023,Z 878.185,A -85,B 0,C 180,E1 -29515.071,E2 -29515.071} C_VEL
LIN {X 0,Y 206.766,Z 876.486,A -85,B 0,C 180,E1 -29517.2,E2 -29517.2} C_VEL
LIN {X 0,Y 206.649,Z 875.72,A -85,B 0,C 180,E1 -29520.001,E2 -29520.001} C_VEL
LIN {X 0,Y 206.663,Z 876.108,A -85,B 0,C 180,E1 -29521.209,E2 -29521.209} C_VEL
LIN {X 0,Y 204.094,Z 892.486,A -85,B 0,C 180,E1 -29521.48,E2 -29521.48} C_VEL
LIN {X 0,Y 200.284,Z 908.337,A -85,B 0,C 180,E1 -29521.732,E2 -29521.732} C_VEL
LIN {X 0,Y 196.236,Z 921.251,A -85,B 0,C 180,E1 -29521.955,E2 -29521.955} C_VEL
LIN {X 0,Y 191.247,Z 934.143,A -85,B 0,C 180,E1 -29522.238,E2 -29522.238} C_VEL
LIN {X 0,Y 185.548,Z 946.448,A -85,B 0,C 180,E1 -29522.587,E2 -29522.587} C_VEL
LIN {X 0,Y 178.589,Z 959.171,A -85,B 0,C 180,E1 -29523.081,E2 -29523.081} C_VEL
LIN {X 0,Y 171.643,Z 970.155,A -85,B 0,C 180,E1 -29523.61,E2 -29523.61} C_VEL
LIN {X 0,Y 163.845,Z 980.938,A -85,B 0,C 180,E1 -29524.238,E2 -29524.238} C_VEL
LIN {X 0,Y 155.219,Z 991.424,A -85,B 0,C 180,E1 -29525.07,E2 -29525.07} C_VEL
LIN {X 0,Y 146.643,Z 1000.687,A -85,B 0,C 180,E1 -29526.046,E2 -29526.046} C_VEL
LIN {X 0,Y 136.381,Z 1010.404,A -85,B 0,C 180,E1 -29527.268,E2 -29527.268} C_VEL
LIN {X 0,Y 126.22,Z 1018.92,A -85,B 0,C 180,E1 -29528.772,E2 -29528.772} C_VEL
LIN {X 0,Y 114.512,Z 1027.515,A -85,B 0,C 180,E1 -29530.903,E2 -29530.903} C_VEL
LIN {X 0,Y 104.63,Z 1033.944,A -85,B 0,C 180,E1 -29533.111,E2 -29533.111} C_VEL
LIN {X 0,Y 91.728,Z 1041.205,A -85,B 0,C 180,E1 -29536.726,E2 -29536.726} C_VEL
LIN {X 0,Y 82.375,Z 1045.861,A -85,B 0,C 180,E1 -29540.205,E2 -29540.205} C_VEL
LIN {X 0,Y 70.518,Z 1050.97,A -85,B 0,C 180,E1 -29546.242,E2 -29546.242} C_VEL
LIN {X 0,Y 59.724,Z 1054.989,A -85,B 0,C 180,E1 -29554.543,E2 -29554.543} C_VEL
LIN {X 0,Y 50.584,Z 1057.97,A -85,B 0,C 180,E1 -29565.999,E2 -29565.999} C_VEL
LIN {X 0,Y 46.921,Z 1059.172,A -85,B 0,C 180,E1 -29573.194,E2 -29573.194} C_VEL
LIN {X 0,Y 42.124,Z 1060.676,A -85,B 0,C 180,E1 -29590.508,E2 -29590.508} C_VEL
LIN {X 0,Y 41.235,Z 1061.198,A -85,B 0,C 180,E1 -29610,E2 -29610} C_VEL
LIN {X 0,Y 42.124,Z 1060.676,A -85,B 0,C 180,E1 -29629.492,E2 -29629.492} C_VEL
LIN {X 0,Y 46.922,Z 1059.172,A -85,B 0,C 180,E1 -29646.806,E2 -29646.806} C_VEL
LIN {X 0,Y 55.037,Z 1056.63,A -85,B 0,C 180,E1 -29660.319,E2 -29660.319} C_VEL
LIN {X 0,Y 67.703,Z 1052.063,A -85,B 0,C 180,E1 -29671.924,E2 -29671.924} C_VEL
LIN {X 0,Y 76.347,Z 1048.563,A -85,B 0,C 180,E1 -29677.001,E2 -29677.001} C_VEL
LIN {X 0,Y 88.577,Z 1042.828,A -85,B 0,C 180,E1 -29682.193,E2 -29682.193} C_VEL
LIN {X 0,Y 98.129,Z 1037.766,A -85,B 0,C 180,E1 -29685.204,E2 -29685.204} C_VEL
LIN {X 0,Y 111.196,Z 1029.736,A -85,B 0,C 180,E1 -29688.417,E2 -29688.417} C_VEL
LIN {X 0,Y 121.181,Z 1022.757,A -85,B 0,C 180,E1 -29690.369,E2 -29690.369} C_VEL
LIN {X 0,Y 131.283,Z 1014.794,A -85,B 0,C 180,E1 -29692.028,E2 -29692.028} C_VEL
LIN {X 0,Y 141.5,Z 1005.694,A -85,B 0,C 180,E1 -29693.379,E2 -29693.379} C_VEL
LIN {X 0,Y 149.928,Z 997.287,A -85,B 0,C 180,E1 -29694.361,E2 -29694.361} C_VEL
LIN {X 0,Y 160.392,Z 985.285,A -85,B 0,C 180,E1 -29695.434,E2 -29695.434} C_VEL
LIN {X 0,Y 169.039,Z 973.888,A -85,B 0,C 180,E1 -29696.201,E2 -29696.201} C_VEL
LIN {X 0,Y 175.984,Z 963.481,A -85,B 0,C 180,E1 -29696.717,E2 -29696.717} C_VEL
LIN {X 0,Y 182.934,Z 951.469,A -85,B 0,C 180,E1 -29697.246,E2 -29697.246} C_VEL
LIN {X 0,Y 189.031,Z 939.162,A -85,B 0,C 180,E1 -29697.651,E2 -29697.651} C_VEL
LIN {X 0,Y 194.463,Z 926.101,A -85,B 0,C 180,E1 -29697.96,E2 -29697.96} C_VEL
LIN {X 0,Y 198.988,Z 912.758,A -85,B 0,C 180,E1 -29698.207,E2 -29698.207} C_VEL
LIN {X 0,Y 202.228,Z 900.86,A -85,B 0,C 180,E1 -29698.386,E2 -29698.386} C_VEL
LIN {X 0,Y 204.972,Z 887.438,A -85,B 0,C 180,E1 -29698.573,E2 -29698.573} C_VEL
LIN {X 0,Y 206.66,Z 876.143,A -85,B 0,C 180,E1 -29698.781,E2 -29698.781} C_VEL
LIN {X 0,Y 206.645,Z 875.761,A -85,B 0,C 180,E1 -29700.487,E2 -29700.487} C_VEL
LIN {X 0,Y 206.826,Z 876.803,A -85,B 0,C 180,E1 -29703.348,E2 -29703.348} C_VEL
LIN {X 0,Y 207.299,Z 879.865,A -85,B 0,C 180,E1 -29706.509,E2 -29706.509} C_VEL
LIN {X 0,Y 207.878,Z 883.496,A -85,B 0,C 180,E1 -29708.934,E2 -29708.934} C_VEL
LIN {X 0,Y 208.608,Z 888.397,A -85,B 0,C 180,E1 -29711.292,E2 -29711.292} C_VEL
LIN {X 0,Y 209.985,Z 898.945,A -85,B 0,C 180,E1 -29715.647,E2 -29715.647} C_VEL
